C09154=1166.613,121.916,-54.152,-178.809,6.458,148.827
C09155=1166.608,122.166,-54.171,-178.807,6.459,148.826
C09156=1166.603,122.415,-54.191,-178.804,6.460,148.826
C09157=1166.598,122.664,-54.210,-178.801,6.462,148.825
C09158=1166.594,122.914,-54.229,-178.798,6.464,148.825
C09159=1166.589,123.163,-54.249,-178.795,6.466,148.825
C09160=1166.584,123.411,-54.269,-178.793,6.467,148.824
C09161=1166.579,123.661,-54.289,-178.790,6.468,148.824
C09162=1166.575,123.911,-54.308,-178.787,6.470,148.823
C09163=1166.569,124.159,-54.328,-178.785,6.471,148.823
C09164=1166.565,124.409,-54.347,-178.782,6.473,148.822
C09165=1166.561,124.658,-54.367,-178.779,6.475,148.822
C09166=1166.556,124.906,-54.386,-178.777,6.477,148.822
C09167=1166.551,125.156,-54.406,-178.773,6.478,148.821
C09168=1166.546,125.406,-54.426,-178.771,6.479,148.821
C09169=1166.541,125.654,-54.445,-178.769,6.481,148.820
C09170=1166.536,125.903,-54.465,-178.766,6.482,148.820
C09171=1166.532,126.153,-54.485,-178.763,6.484,148.819
C09172=1166.527,126.403,-54.505,-178.760,6.486,148.819
C09173=1166.522,126.651,-54.525,-178.757,6.487,148.818
C09174=1166.517,126.900,-54.544,-178.755,6.488,148.818
C09175=1166.512,127.150,-54.564,-178.752,6.490,148.817
C09176=1166.507,127.399,-54.583,-178.750,6.491,148.817
C09177=1166.502,127.648,-54.604,-178.747,6.493,148.817
C09178=1166.498,127.897,-54.623,-178.744,6.495,148.816
C09179=1166.493,128.147,-54.643,-178.741,6.496,148.816
C09180=1166.488,128.395,-54.663,-178.738,6.498,148.815
C09181=1166.483,128.645,-54.683,-178.736,6.500,148.815
C09182=1166.479,128.894,-54.703,-178.733,6.501,148.814
C09183=1166.474,129.143,-54.723,-178.731,6.502,148.814
C09184=1166.469,129.392,-54.742,-178.728,6.504,148.814
C09185=1166.464,129.641,-54.762,-178.725,6.506,148.813
C09186=1166.460,129.891,-54.782,-178.722,6.507,148.813
C09187=1166.455,130.140,-54.802,-178.719,6.509,148.812
C09188=1166.450,130.389,-54.822,-178.717,6.511,148.812
C09189=1166.445,130.637,-54.842,-178.714,6.512,148.812
C09190=1166.441,130.887,-54.862,-178.712,6.513,148.811
C09191=1166.436,131.136,-54.882,-178.709,6.515,148.811
C09192=1166.431,131.385,-54.902,-178.707,6.517,148.810
C09193=1166.427,131.634,-54.922,-178.704,6.519,148.810
C09194=1166.421,131.903,-54.943,-178.701,6.520,148.809
C09195=1166.416,132.171,-54.965,-178.698,6.522,148.809
C09196=1166.410,132.440,-54.987,-178.695,6.524,148.809
C09197=1166.406,132.708,-55.008,-178.691,6.526,148.808
C09198=1166.401,132.958,-55.028,-178.689,6.527,148.808
C09199=1166.396,133.207,-55.048,-178.687,6.528,148.807
C09200=1166.391,133.456,-55.069,-178.684,6.530,148.807
C09201=1166.386,133.706,-55.089,-178.681,6.532,148.806
C09202=1166.382,133.955,-55.109,-178.679,6.533,148.806
C09203=1166.377,134.204,-55.129,-178.676,6.535,148.806
C09204=1166.372,134.452,-55.149,-178.673,6.537,148.805
C09205=1166.368,134.701,-55.169,-178.670,6.538,148.805
C09206=1166.362,134.951,-55.189,-178.667,6.540,148.804
C09207=1166.358,135.200,-55.210,-178.665,6.542,148.804
C09208=1166.353,135.449,-55.230,-178.662,6.543,148.803
C09209=1166.349,135.699,-55.250,-178.659,6.545,148.803
C09210=1166.344,135.948,-55.270,-178.656,6.547,148.803
C09211=1166.339,136.197,-55.291,-178.654,6.548,148.802
C09212=1166.334,136.446,-55.310,-178.652,6.550,148.802
C09213=1166.329,136.695,-55.331,-178.649,6.551,148.801
C09214=1166.325,136.944,-55.351,-178.646,6.553,148.801
C09215=1166.320,137.193,-55.372,-178.643,6.554,148.800
C09216=1166.315,137.442,-55.392,-178.640,6.556,148.800
C09217=1166.310,137.691,-55.412,-178.638,6.558,148.800
C09218=1166.305,137.941,-55.433,-178.635,6.560,148.799
C09219=1166.301,138.190,-55.453,-178.632,6.561,148.799
C09220=1166.296,138.439,-55.473,-178.629,6.563,148.798
C09221=1166.292,138.688,-55.493,-178.627,6.565,148.798
C09222=1166.287,138.937,-55.514,-178.624,6.567,148.798
C09223=1166.282,139.186,-55.535,-178.621,6.568,148.797
C09224=1166.278,139.435,-55.555,-178.619,6.570,148.797
C09225=1166.272,139.685,-55.576,-178.616,6.572,148.797
C09226=1166.268,139.934,-55.597,-178.613,6.573,148.796
C09227=1166.263,140.183,-55.616,-178.611,6.574,148.796
C09228=1166.258,140.432,-55.637,-178.608,6.576,148.795
C09229=1166.254,140.681,-55.658,-178.605,6.578,148.795
C09230=1166.249,140.930,-55.678,-178.603,6.579,148.794
C09231=1166.244,141.180,-55.699,-178.600,6.581,148.794
C09232=1166.240,141.428,-55.719,-178.597,6.583,148.794
C09233=1166.234,141.678,-55.740,-178.594,6.584,148.793
C09234=1166.230,141.927,-55.761,-178.592,6.586,148.793
C09235=1166.226,142.176,-55.781,-178.589,6.588,148.792
C09236=1166.220,142.425,-55.802,-178.586,6.590,148.792
C09237=1166.216,142.674,-55.822,-178.584,6.591,148.792
C09238=1166.211,142.923,-55.843,-178.581,6.593,148.791
C09239=1166.206,143.172,-55.864,-178.578,6.595,148.791
C09240=1166.202,143.421,-55.884,-178.576,6.597,148.791
C09241=1166.197,143.670,-55.905,-178.573,6.598,148.790
C09242=1166.192,143.919,-55.925,-178.570,6.600,148.790
C09243=1166.187,144.168,-55.946,-178.567,6.601,148.789
C09244=1166.183,144.417,-55.967,-178.564,6.603,148.789
C09245=1166.178,144.667,-55.988,-178.562,6.605,148.788
C09246=1166.173,144.916,-56.008,-178.559,6.607,148.788
C09247=1166.168,145.165,-56.029,-178.556,6.608,148.788
C09248=1166.163,145.414,-56.049,-178.553,6.610,148.787
C09249=1166.158,145.663,-56.070,-178.551,6.612,148.787
C09250=1166.154,145.911,-56.091,-178.548,6.614,148.786
C09251=1166.149,146.161,-56.112,-178.545,6.615,148.786
C09252=1166.145,146.410,-56.133,-178.543,6.617,148.786
C09253=1166.140,146.660,-56.154,-178.540,6.619,148.785
C09254=1166.136,146.909,-56.174,-178.537,6.621,148.785
C09255=1166.130,147.158,-56.195,-178.535,6.622,148.785
C09256=1166.125,147.406,-56.217,-178.532,6.624,148.784
C09257=1166.121,147.655,-56.237,-178.529,6.626,148.784
C09258=1166.116,147.905,-56.258,-178.526,6.628,148.783
C09259=1166.111,148.154,-56.279,-178.524,6.629,148.783
C09260=1166.106,148.403,-56.300,-178.521,6.631,148.783
C09261=1166.102,148.652,-56.322,-178.518,6.633,148.782
C09262=1166.098,148.901,-56.342,-178.516,6.635,148.782
C09263=1166.092,149.150,-56.363,-178.513,6.636,148.781
C09264=1166.088,149.399,-56.384,-178.510,6.638,148.781
C09265=1166.083,149.648,-56.405,-178.508,6.640,148.781
C09266=1166.078,149.897,-56.426,-178.505,6.642,148.780
C09267=1166.073,150.146,-56.447,-178.502,6.643,148.780
C09268=1166.069,150.396,-56.469,-178.499,6.645,148.780
C09269=1166.064,150.645,-56.490,-178.497,6.647,148.779
C09270=1166.060,150.894,-56.510,-178.494,6.648,148.779
C09271=1166.055,151.142,-56.532,-178.491,6.650,148.778
C09272=1166.050,151.392,-56.553,-178.489,6.652,148.778
C09273=1166.045,151.640,-56.574,-178.486,6.654,148.778
C09274=1166.041,151.890,-56.595,-178.483,6.655,148.777
C09275=1166.036,152.139,-56.616,-178.481,6.657,148.777
C09276=1166.031,152.388,-56.638,-178.478,6.659,148.777
C09277=1166.026,152.637,-56.658,-178.475,6.661,148.776
C09278=1166.021,152.885,-56.680,-178.473,6.662,148.776
C09279=1166.017,153.135,-56.701,-178.469,6.665,148.775
C09280=1166.013,153.384,-56.722,-178.467,6.667,148.775
C09281=1166.008,153.633,-56.743,-178.464,6.668,148.775
C09282=1166.002,153.882,-56.764,-178.461,6.670,148.774
C09283=1165.998,154.132,-56.786,-178.458,6.672,148.774
C09284=1165.993,154.381,-56.807,-178.456,6.674,148.774
C09285=1165.989,154.629,-56.828,-178.453,6.675,148.773
C09286=1165.984,154.878,-56.849,-178.450,6.677,148.773
C09287=1165.979,155.128,-56.871,-178.448,6.679,148.772
C09288=1165.975,155.376,-56.893,-178.445,6.681,148.772
C09289=1165.969,155.626,-56.914,-178.442,6.682,148.772
C09290=1165.965,155.874,-56.935,-178.440,6.684,148.771
C09291=1165.961,156.124,-56.956,-178.437,6.686,148.771
C09292=1165.956,156.373,-56.978,-178.434,6.688,148.771
C09293=1165.951,156.622,-56.999,-178.431,6.689,148.770
C09294=1165.946,156.871,-57.021,-178.429,6.691,148.770
C09295=1165.941,157.120,-57.043,-178.426,6.694,148.769
C09296=1165.937,157.369,-57.063,-178.423,6.695,148.769
C09297=1165.932,157.617,-57.085,-178.420,6.697,148.769
C09298=1165.927,157.887,-57.108,-178.417,6.699,148.768
C09299=1165.922,158.155,-57.132,-178.415,6.701,148.768
C09300=1165.917,158.425,-57.155,-178.411,6.703,148.768
C09301=1165.912,158.694,-57.178,-178.409,6.705,148.767
C09302=1165.907,158.942,-57.199,-178.406,6.707,148.767
C09303=1165.903,159.192,-57.221,-178.403,6.709,148.766
C09304=1165.898,159.441,-57.242,-178.401,6.710,148.766
C09305=1165.893,159.690,-57.264,-178.398,6.712,148.766
C09306=1165.889,159.939,-57.286,-178.395,6.714,148.765
C09307=1165.884,160.187,-57.308,-178.392,6.716,148.765
C09308=1165.879,160.437,-57.329,-178.389,6.718,148.765
C09309=1165.874,160.686,-57.351,-178.387,6.720,148.764
C09310=1165.869,160.935,-57.372,-178.384,6.722,148.764
C09311=1165.865,161.184,-57.394,-178.382,6.724,148.764
C09312=1165.860,161.433,-57.416,-178.379,6.725,148.763
C09313=1165.855,161.682,-57.437,-178.376,6.727,148.763
C09314=1165.851,161.931,-57.459,-178.374,6.729,148.763
C09315=1165.846,162.180,-57.481,-178.371,6.731,148.762
C09316=1165.842,162.429,-57.503,-178.368,6.733,148.762
C09317=1165.837,162.678,-57.525,-178.365,6.735,148.761
C09318=1165.833,162.927,-57.547,-178.362,6.737,148.761
C09319=1165.828,163.176,-57.568,-178.360,6.738,148.761
C09320=1165.823,163.425,-57.590,-178.357,6.740,148.760
C09321=1165.819,163.674,-57.612,-178.354,6.742,148.760
C09322=1165.814,163.923,-57.634,-178.352,6.744,148.760
C09323=1165.809,164.172,-57.655,-178.349,6.746,148.759
C09324=1165.804,164.421,-57.677,-178.347,6.748,148.759
C09325=1165.800,164.670,-57.699,-178.343,6.750,148.759
C09326=1165.795,164.919,-57.720,-178.341,6.752,148.758
C09327=1165.790,165.168,-57.742,-178.338,6.754,148.758
C09328=1165.785,165.417,-57.765,-178.335,6.755,148.758
C09329=1165.780,165.666,-57.786,-178.333,6.757,148.757
C09330=1165.776,165.915,-57.809,-178.330,6.759,148.757
C09331=1165.771,166.164,-57.830,-178.327,6.761,148.756
C09332=1165.767,166.413,-57.853,-178.324,6.763,148.756
C09333=1165.762,166.661,-57.875,-178.322,6.765,148.756
C09334=1165.758,166.911,-57.897,-178.319,6.767,148.756
C09335=1165.752,167.160,-57.919,-178.316,6.769,148.755
C09336=1165.748,167.409,-57.941,-178.314,6.771,148.755
C09337=1165.743,167.658,-57.963,-178.311,6.772,148.754
C09338=1165.739,167.907,-57.985,-178.308,6.774,148.754
C09339=1165.734,168.156,-58.006,-178.305,6.777,148.754
C09340=1165.729,168.405,-58.029,-178.302,6.778,148.753
C09341=1165.725,168.653,-58.051,-178.300,6.781,148.753
C09342=1165.720,168.903,-58.074,-178.297,6.782,148.753
C09343=1165.716,169.151,-58.095,-178.295,6.784,148.753
C09344=1165.711,169.401,-58.118,-178.292,6.786,148.752
C09345=1165.706,169.650,-58.140,-178.289,6.788,148.752
C09346=1165.701,169.899,-58.162,-178.286,6.790,148.751
C09347=1165.697,170.148,-58.184,-178.283,6.792,148.751
C09348=1165.692,170.397,-58.207,-178.281,6.794,148.751
C09349=1165.688,170.646,-58.229,-178.279,6.796,148.751
C09350=1165.683,170.895,-58.250,-178.276,6.797,148.750
C09351=1165.679,171.143,-58.273,-178.273,6.800,148.750
C09352=1165.673,171.392,-58.295,-178.270,6.802,148.749
C09353=1165.669,171.642,-58.317,-178.267,6.804,148.749
C09354=1165.665,171.890,-58.340,-178.265,6.805,148.749
C09355=1165.659,172.139,-58.363,-178.262,6.807,148.748
C09356=1165.655,172.389,-58.385,-178.259,6.810,148.748
C09357=1165.650,172.637,-58.407,-178.256,6.812,148.748
C09358=1165.645,172.886,-58.430,-178.254,6.814,148.748
C09359=1165.641,173.136,-58.452,-178.251,6.815,148.747
C09360=1165.637,173.384,-58.474,-178.248,6.817,148.747
C09361=1165.632,173.633,-58.497,-178.245,6.820,148.746
C09362=1165.627,173.882,-58.518,-178.243,6.822,148.746
C09363=1165.622,174.131,-58.542,-178.240,6.823,148.746
C09364=1165.618,174.380,-58.564,-178.237,6.825,148.746
C09365=1165.613,174.628,-58.586,-178.235,6.827,148.745
C09366=1165.608,174.878,-58.609,-178.231,6.830,148.745
C09367=1165.604,175.127,-58.632,-178.229,6.831,148.744
C09368=1165.599,175.376,-58.654,-178.227,6.833,148.744
C09369=1165.595,175.624,-58.677,-178.224,6.835,148.744
C09370=1165.590,175.874,-58.699,-178.221,6.837,148.744
C09371=1165.585,176.123,-58.721,-178.218,6.840,148.743
C09372=1165.581,176.371,-58.744,-178.215,6.841,148.743
C09373=1165.576,176.620,-58.767,-178.213,6.843,148.743
C09374=1165.571,176.869,-58.789,-178.210,6.845,148.742
C09375=1165.567,177.118,-58.812,-178.208,6.847,148.742
C09376=1165.562,177.367,-58.834,-178.204,6.849,148.742
C09377=1165.557,177.616,-58.857,-178.202,6.851,148.741
C09378=1165.553,177.865,-58.879,-178.200,6.853,148.741
C09379=1165.548,178.114,-58.903,-178.197,6.855,148.741
C09380=1165.544,178.363,-58.925,-178.194,6.858,148.740
C09381=1165.538,178.612,-58.948,-178.191,6.859,148.740
C09382=1165.534,178.861,-58.970,-178.188,6.861,148.740
C09383=1165.529,179.110,-58.993,-178.186,6.863,148.740
C09384=1165.525,179.358,-59.015,-178.183,6.866,148.739
C09385=1165.520,179.607,-59.039,-178.180,6.868,148.739
C09386=1165.516,179.857,-59.061,-178.177,6.869,148.739
C09387=1165.511,180.106,-59.084,-178.175,6.871,148.738
C09388=1165.506,180.354,-59.107,-178.172,6.873,148.738
C09389=1165.502,180.603,-59.130,-178.169,6.876,148.738
C09390=1165.497,180.852,-59.153,-178.167,6.878,148.737
C09391=1165.493,181.101,-59.175,-178.164,6.879,148.737
C09392=1165.488,181.350,-59.199,-178.161,6.881,148.737
C09393=1165.483,181.599,-59.221,-178.158,6.884,148.737
C09394=1165.479,181.848,-59.244,-178.156,6.886,148.736
C09395=1165.474,182.097,-59.267,-178.153,6.888,148.736
C09396=1165.470,182.345,-59.290,-178.150,6.889,148.735
C09397=1165.465,182.595,-59.313,-178.148,6.892,148.735
C09398=1165.460,182.843,-59.335,-178.145,6.894,148.735
C09399=1165.456,183.092,-59.358,-178.142,6.896,148.735
C09400=1165.451,183.341,-59.382,-178.139,6.898,148.734
C09401=1165.446,183.590,-59.405,-178.137,6.900,148.734
C09402=1165.442,183.860,-59.429,-178.134,6.902,148.734
C09403=1165.437,184.129,-59.454,-178.131,6.905,148.733
C09404=1165.431,184.399,-59.479,-178.128,6.907,148.733
C09405=1165.427,184.668,-59.505,-178.125,6.909,148.733
C09406=1165.422,184.918,-59.527,-178.122,6.911,148.732
C09407=1165.417,185.167,-59.551,-178.119,6.914,148.732
C09408=1165.412,185.415,-59.574,-178.117,6.916,148.732
C09409=1165.408,185.664,-59.596,-178.114,6.917,148.732
C09410=1165.403,185.913,-59.620,-178.111,6.919,148.731
C09411=1165.399,186.162,-59.643,-178.109,6.922,148.731
C09412=1165.394,186.411,-59.666,-178.106,6.924,148.731
C09413=1165.390,186.660,-59.689,-178.103,6.926,148.730
C09414=1165.385,186.909,-59.713,-178.100,6.928,148.730
C09415=1165.380,187.158,-59.736,-178.098,6.930,148.730
C09416=1165.376,187.407,-59.759,-178.095,6.932,148.730
C09417=1165.370,187.655,-59.782,-178.092,6.934,148.729
C09418=1165.367,187.904,-59.805,-178.089,6.936,148.729
C09419=1165.362,188.153,-59.828,-178.087,6.938,148.729
C09420=1165.357,188.401,-59.853,-178.084,6.940,148.728
C09421=1165.353,188.650,-59.876,-178.081,6.943,148.728
C09422=1165.348,188.899,-59.899,-178.079,6.945,148.728
C09423=1165.343,189.148,-59.923,-178.076,6.947,148.728
C09424=1165.339,189.397,-59.946,-178.073,6.949,148.727
C09425=1165.335,189.646,-59.969,-178.070,6.951,148.727
C09426=1165.330,189.895,-59.992,-178.068,6.953,148.727
C09427=1165.325,190.144,-60.015,-178.065,6.956,148.726
C09428=1165.321,190.393,-60.039,-178.062,6.958,148.726
C09429=1165.316,190.642,-60.063,-178.060,6.960,148.726
C09430=1165.311,190.891,-60.086,-178.057,6.961,148.726
C09431=1165.306,191.139,-60.109,-178.054,6.964,148.725
C09432=1165.301,191.388,-60.133,-178.052,6.966,148.725
C09433=1165.297,191.636,-60.157,-178.049,6.968,148.725
C09434=1165.292,191.885,-60.180,-178.046,6.970,148.724
C09435=1165.288,192.134,-60.203,-178.043,6.972,148.724
C09436=1165.283,192.383,-60.227,-178.041,6.974,148.724
C09437=1165.279,192.632,-60.251,-178.038,6.977,148.724
C09438=1165.274,192.881,-60.274,-178.035,6.979,148.723
C09439=1165.269,193.130,-60.298,-178.033,6.981,148.723
C09440=1165.265,193.378,-60.322,-178.029,6.983,148.723
C09441=1165.260,193.627,-60.345,-178.027,6.985,148.722
C09442=1165.255,193.876,-60.368,-178.025,6.987,148.722
C09443=1165.251,194.125,-60.392,-178.021,6.990,148.722
C09444=1165.246,194.374,-60.416,-178.019,6.992,148.722
C09445=1165.242,194.624,-60.439,-178.016,6.995,148.721
C09446=1165.238,194.872,-60.464,-178.013,6.996,148.721
C09447=1165.233,195.121,-60.487,-178.010,6.998,148.721
C09448=1165.229,195.369,-60.511,-178.008,7.001,148.721
C09449=1165.224,195.619,-60.534,-178.005,7.003,148.720
C09450=1165.219,195.868,-60.558,-178.002,7.005,148.720
C09451=1165.215,196.116,-60.582,-178.000,7.007,148.720
C09452=1165.210,196.365,-60.605,-177.997,7.009,148.720
C09453=1165.206,196.613,-60.629,-177.994,7.011,148.719
C09454=1165.201,196.862,-60.653,-177.991,7.014,148.719
C09455=1165.197,197.111,-60.677,-177.989,7.016,148.719
C09456=1165.191,197.360,-60.701,-177.987,7.018,148.719
C09457=1165.187,197.609,-60.725,-177.983,7.020,148.718
C09458=1165.182,197.858,-60.748,-177.981,7.022,148.718
C09459=1165.178,198.107,-60.772,-177.978,7.025,148.718
C09460=1165.174,198.356,-60.796,-177.975,7.027,148.717
C09461=1165.169,198.604,-60.820,-177.972,7.029,148.717
C09462=1165.165,198.853,-60.844,-177.970,7.032,148.717
C09463=1165.159,199.102,-60.868,-177.967,7.033,148.717
C09464=1165.155,199.350,-60.892,-177.964,7.035,148.716
C09465=1165.150,199.599,-60.915,-177.962,7.038,148.716
C09466=1165.147,199.849,-60.940,-177.959,7.040,148.716
C09467=1165.142,200.097,-60.964,-177.956,7.043,148.716
C09468=1165.137,200.346,-60.988,-177.953,7.045,148.715
C09469=1165.132,200.595,-61.012,-177.951,7.046,148.715
C09470=1165.128,200.843,-61.036,-177.948,7.049,148.715
C09471=1165.123,201.092,-61.059,-177.945,7.051,148.715
C09472=1165.119,201.342,-61.084,-177.943,7.054,148.715
C09473=1165.114,201.590,-61.108,-177.940,7.056,148.714
C09474=1165.110,201.839,-61.132,-177.937,7.058,148.714
C09475=1165.105,202.087,-61.156,-177.934,7.060,148.714
C09476=1165.100,202.336,-61.181,-177.932,7.062,148.713
C09477=1165.096,202.585,-61.205,-177.928,7.065,148.713
C09478=1165.092,202.834,-61.229,-177.926,7.067,148.713
C09479=1165.087,203.083,-61.252,-177.924,7.069,148.713
C09480=1165.082,203.331,-61.277,-177.921,7.072,148.712
C09481=1165.078,203.580,-61.301,-177.918,7.073,148.712
C09482=1165.074,203.829,-61.326,-177.915,7.076,148.712
C09483=1165.069,204.078,-61.350,-177.913,7.078,148.712
C09484=1165.064,204.327,-61.374,-177.909,7.081,148.711
C09485=1165.060,204.575,-61.398,-177.907,7.083,148.711
C09486=1165.055,204.825,-61.423,-177.905,7.085,148.711
C09487=1165.051,205.073,-61.447,-177.902,7.088,148.711
C09488=1165.046,205.321,-61.471,-177.899,7.089,148.710
C09489=1165.041,205.570,-61.496,-177.896,7.092,148.710
C09490=1165.037,205.819,-61.520,-177.894,7.094,148.710
C09491=1165.032,206.068,-61.545,-177.891,7.096,148.710
C09492=1165.028,206.316,-61.569,-177.888,7.099,148.710
C09493=1165.023,206.565,-61.593,-177.886,7.101,148.709
C09494=1165.019,206.814,-61.618,-177.883,7.103,148.709
C09495=1165.015,207.063,-61.642,-177.880,7.105,148.709
C09496=1165.009,207.311,-61.667,-177.877,7.108,148.708
C09497=1165.006,207.560,-61.691,-177.875,7.110,148.708
C09498=1165.001,207.809,-61.716,-177.871,7.113,148.708
C09499=1164.996,208.058,-61.740,-177.869,7.115,148.708
C09500=1164.991,208.306,-61.764,-177.867,7.116,148.708
C09501=1164.987,208.555,-61.789,-177.864,7.119,148.707
C09502=1164.982,208.804,-61.814,-177.861,7.121,148.707
C09503=1164.978,209.053,-61.838,-177.858,7.124,148.707
C09504=1164.973,209.302,-61.863,-177.856,7.126,148.707
C09505=1164.969,209.550,-61.887,-177.853,7.129,148.707
C09506=1164.964,209.821,-61.913,-177.850,7.131,148.706
C09507=1164.959,210.091,-61.941,-177.847,7.133,148.706
C09508=1164.954,210.362,-61.967,-177.844,7.136,148.706
C09509=1164.949,210.632,-61.994,-177.841,7.139,148.705
C09510=1164.944,210.881,-62.019,-177.838,7.140,148.705
C09511=1164.940,211.130,-62.043,-177.836,7.143,148.705
C09512=1164.935,211.379,-62.068,-177.833,7.145,148.705
C09513=1164.931,211.627,-62.092,-177.830,7.148,148.705
C09514=1164.927,211.876,-62.118,-177.827,7.150,148.704
C09515=1164.922,212.125,-62.143,-177.825,7.153,148.704
C09516=1164.917,212.373,-62.167,-177.822,7.155,148.704
C09517=1164.913,212.623,-62.192,-177.819,7.158,148.704
C09518=1164.909,212.871,-62.216,-177.817,7.159,148.703
C09519=1164.904,213.120,-62.242,-177.814,7.162,148.703
C09520=1164.899,213.369,-62.266,-177.811,7.164,148.703
C09521=1164.894,213.617,-62.290,-177.809,7.166,148.703
C09522=1164.890,213.866,-62.316,-177.806,7.169,148.703
C09523=1164.885,214.115,-62.341,-177.803,7.171,148.702
C09524=1164.881,214.364,-62.365,-177.800,7.174,148.702
C09525=1164.877,214.612,-62.391,-177.798,7.176,148.702
C09526=1164.872,214.861,-62.416,-177.795,7.178,148.702
C09527=1164.868,215.110,-62.440,-177.793,7.180,148.702
C09528=1164.863,215.359,-62.465,-177.789,7.183,148.701
C09529=1164.858,215.607,-62.490,-177.787,7.185,148.701
C09530=1164.853,215.855,-62.515,-177.784,7.188,148.701
C09531=1164.850,216.104,-62.540,-177.782,7.190,148.701
C09532=1164.845,216.353,-62.565,-177.778,7.192,148.700
C09533=1164.840,216.602,-62.590,-177.776,7.194,148.700
C09534=1164.835,216.851,-62.615,-177.773,7.197,148.700
C09535=1164.832,217.099,-62.640,-177.770,7.200,148.700
C09536=1164.827,217.348,-62.665,-177.768,7.202,148.700
C09537=1164.822,217.597,-62.691,-177.765,7.205,148.699
C09538=1164.817,217.845,-62.715,-177.762,7.207,148.699
C09539=1164.814,218.094,-62.740,-177.759,7.209,148.699
C09540=1164.809,218.343,-62.765,-177.757,7.211,148.699
C09541=1164.804,218.591,-62.791,-177.754,7.214,148.699
C09542=1164.800,218.840,-62.817,-177.752,7.216,148.698
C09543=1164.795,219.089,-62.841,-177.748,7.219,148.698
C09544=1164.791,219.338,-62.866,-177.746,7.221,148.698
C09545=1164.786,219.586,-62.891,-177.743,7.224,148.698
C09546=1164.782,219.835,-62.917,-177.741,7.226,148.698
C09547=1164.777,220.083,-62.942,-177.738,7.228,148.697
C09548=1164.773,220.333,-62.967,-177.735,7.230,148.697
C09549=1164.768,220.581,-62.993,-177.732,7.233,148.697
C09550=1164.764,220.829,-63.018,-177.730,7.235,148.697
C09551=1164.760,221.079,-63.043,-177.727,7.238,148.697
C09552=1164.755,221.327,-63.068,-177.724,7.241,148.696
C09553=1164.751,221.575,-63.094,-177.722,7.243,148.696
C09554=1164.746,221.824,-63.119,-177.718,7.245,148.696
C09555=1164.742,222.073,-63.144,-177.716,7.248,148.696
C09556=1164.737,222.322,-63.170,-177.713,7.250,148.696
C09557=1164.732,222.570,-63.195,-177.711,7.252,148.695
C09558=1164.728,222.819,-63.221,-177.708,7.255,148.695
C09559=1164.723,223.067,-63.246,-177.705,7.257,148.695
C09560=1164.719,223.316,-63.272,-177.703,7.260,148.695
C09561=1164.715,223.565,-63.297,-177.699,7.263,148.695
C09562=1164.710,223.814,-63.322,-177.697,7.265,148.695
C09563=1164.705,224.063,-63.348,-177.694,7.267,148.694
C09564=1164.701,224.311,-63.374,-177.692,7.269,148.694
C09565=1164.696,224.560,-63.399,-177.689,7.272,148.694
C09566=1164.692,224.808,-63.425,-177.686,7.274,148.694
C09567=1164.687,225.056,-63.450,-177.684,7.277,148.694
C09568=1164.683,225.305,-63.476,-177.680,7.280,148.693
C09569=1164.678,225.555,-63.501,-177.678,7.282,148.693
C09570=1164.674,225.803,-63.526,-177.675,7.285,148.693
C09571=1164.669,226.052,-63.552,-177.673,7.287,148.693
C09572=1164.665,226.300,-63.578,-177.670,7.290,148.693
C09573=1164.661,226.549,-63.604,-177.667,7.291,148.692
C09574=1164.656,226.797,-63.629,-177.665,7.294,148.692
C09575=1164.652,227.046,-63.655,-177.662,7.297,148.692
C09576=1164.648,227.295,-63.680,-177.659,7.299,148.692
C09577=1164.642,227.543,-63.706,-177.656,7.302,148.692
C09578=1164.638,227.792,-63.732,-177.654,7.304,148.692
C09579=1164.634,228.041,-63.758,-177.651,7.307,148.691
C09580=1164.629,228.290,-63.784,-177.648,7.310,148.691
C09581=1164.625,228.538,-63.809,-177.645,7.311,148.691
C09582=1164.620,228.787,-63.835,-177.643,7.314,148.691
C09583=1164.616,229.035,-63.861,-177.640,7.316,148.691
C09584=1164.611,229.284,-63.886,-177.637,7.319,148.690
C09585=1164.607,229.532,-63.913,-177.634,7.322,148.690
C09586=1164.602,229.781,-63.939,-177.632,7.324,148.690
C09587=1164.598,230.030,-63.964,-177.629,7.327,148.690
C09588=1164.594,230.278,-63.990,-177.626,7.330,148.690
C09589=1164.588,230.527,-64.016,-177.624,7.332,148.690
C09590=1164.584,230.776,-64.042,-177.621,7.334,148.689
C09591=1164.580,231.024,-64.068,-177.619,7.337,148.689
C09592=1164.576,231.273,-64.094,-177.615,7.339,148.689
C09593=1164.571,231.521,-64.120,-177.613,7.342,148.689
C09594=1164.566,231.770,-64.146,-177.610,7.344,148.689
C09595=1164.562,232.019,-64.172,-177.607,7.347,148.689
C09596=1164.558,232.267,-64.197,-177.604,7.350,148.689
C09597=1164.554,232.516,-64.224,-177.602,7.352,148.688
C09598=1164.548,232.764,-64.250,-177.599,7.355,148.688
C09599=1164.544,233.013,-64.276,-177.597,7.357,148.688
C09600=1164.540,233.261,-64.302,-177.594,7.360,148.688
C09601=1164.535,233.510,-64.328,-177.591,7.363,148.688
C09602=1164.531,233.759,-64.354,-177.589,7.364,148.688
C09603=1164.527,234.008,-64.380,-177.586,7.367,148.687
C09604=1164.522,234.256,-64.407,-177.583,7.370,148.687
C09605=1164.517,234.504,-64.432,-177.580,7.372,148.687
C09606=1164.513,234.753,-64.459,-177.578,7.375,148.687
C09607=1164.508,235.002,-64.485,-177.575,7.378,148.687
C09608=1164.504,235.250,-64.511,-177.572,7.380,148.687
C09609=1164.500,235.499,-64.537,-177.570,7.383,148.686
C09610=1164.495,235.771,-64.566,-177.567,7.386,148.686
C09611=1164.490,236.042,-64.595,-177.564,7.388,148.686
C09612=1164.485,236.314,-64.623,-177.561,7.391,148.686
C09613=1164.481,236.586,-64.652,-177.558,7.394,148.686
C09614=1164.476,236.835,-64.679,-177.555,7.397,148.686
C09615=1164.472,237.083,-64.705,-177.553,7.399,148.686
C09616=1164.467,237.331,-64.730,-177.550,7.402,148.685
C09617=1164.462,237.580,-64.757,-177.547,7.404,148.685
C09618=1164.458,237.828,-64.783,-177.544,7.407,148.685
C09619=1164.453,238.077,-64.810,-177.542,7.409,148.685
C09620=1164.449,238.326,-64.836,-177.538,7.412,148.685
C09621=1164.445,238.574,-64.863,-177.536,7.414,148.685
C09622=1164.441,238.822,-64.890,-177.533,7.417,148.685
C09623=1164.436,239.071,-64.916,-177.531,7.420,148.684
C09624=1164.432,239.320,-64.942,-177.528,7.422,148.684
C09625=1164.427,239.569,-64.969,-177.525,7.425,148.684
C09626=1164.423,239.817,-64.995,-177.522,7.428,148.684
C09627=1164.418,240.065,-65.022,-177.520,7.430,148.684
C09628=1164.414,240.314,-65.048,-177.517,7.433,148.684
C09629=1164.409,240.563,-65.075,-177.514,7.435,148.684
C09630=1164.405,240.811,-65.101,-177.512,7.438,148.683
C09631=1164.400,241.060,-65.128,-177.509,7.441,148.683
C09632=1164.396,241.309,-65.155,-177.506,7.443,148.683
C09633=1164.392,241.557,-65.181,-177.503,7.446,148.683
C09634=1164.387,241.806,-65.208,-177.501,7.448,148.683
C09635=1164.383,242.054,-65.234,-177.498,7.451,148.683
C09636=1164.378,242.303,-65.261,-177.496,7.454,148.683
C09637=1164.374,242.551,-65.288,-177.493,7.456,148.682
C09638=1164.370,242.799,-65.315,-177.490,7.459,148.682
C09639=1164.365,243.048,-65.341,-177.487,7.462,148.682
C09640=1164.361,243.297,-65.368,-177.485,7.465,148.682
C09641=1164.356,243.545,-65.395,-177.482,7.467,148.682
C09642=1164.352,243.793,-65.422,-177.479,7.470,148.682
C09643=1164.348,244.042,-65.448,-177.476,7.473,148.682
C09644=1164.343,244.291,-65.474,-177.474,7.475,148.682
C09645=1164.338,244.539,-65.502,-177.472,7.478,148.682
C09646=1164.334,244.787,-65.528,-177.468,7.480,148.681
C09647=1164.329,245.036,-65.555,-177.466,7.483,148.681
C09648=1164.325,245.284,-65.582,-177.463,7.485,148.681
C09649=1164.321,245.533,-65.609,-177.461,7.488,148.681
C09650=1164.317,245.782,-65.636,-177.458,7.491,148.681
C09651=1164.312,246.030,-65.663,-177.455,7.494,148.681
C09652=1164.307,246.279,-65.690,-177.452,7.496,148.681
C09653=1164.304,246.527,-65.717,-177.450,7.499,148.681
C09654=1164.299,246.776,-65.744,-177.447,7.502,148.680
C09655=1164.294,247.024,-65.771,-177.445,7.504,148.680
C09656=1164.290,247.273,-65.798,-177.442,7.507,148.680
C09657=1164.286,247.521,-65.824,-177.439,7.510,148.680
C09658=1164.281,247.769,-65.851,-177.436,7.512,148.680
C09659=1164.277,248.018,-65.879,-177.434,7.515,148.680
C09660=1164.272,248.267,-65.906,-177.431,7.518,148.680
C09661=1164.268,248.515,-65.933,-177.428,7.521,148.680
C09662=1164.264,248.764,-65.959,-177.425,7.523,148.680
C09663=1164.259,249.012,-65.986,-177.423,7.525,148.679
C09664=1164.254,249.261,-66.013,-177.420,7.528,148.679
C09665=1164.250,249.509,-66.041,-177.417,7.531,148.679
C09666=1164.246,249.758,-66.069,-177.415,7.534,148.679
C09667=1164.241,250.006,-66.096,-177.412,7.536,148.679
C09668=1164.237,250.255,-66.123,-177.410,7.539,148.679
C09669=1164.233,250.503,-66.149,-177.407,7.542,148.679
C09670=1164.228,250.751,-66.176,-177.404,7.545,148.679
C09671=1164.224,251.000,-66.204,-177.401,7.548,148.679
C09672=1164.220,251.248,-66.232,-177.399,7.550,148.678
C09673=1164.215,251.497,-66.259,-177.396,7.553,148.678
C09674=1164.210,251.745,-66.286,-177.393,7.556,148.678
C09675=1164.206,251.994,-66.313,-177.390,7.559,148.678
C09676=1164.202,252.242,-66.341,-177.388,7.561,148.678
C09677=1164.197,252.491,-66.368,-177.385,7.564,148.678
C09678=1164.193,252.739,-66.395,-177.382,7.566,148.678
C09679=1164.188,252.988,-66.422,-177.379,7.569,148.678
C09680=1164.184,253.236,-66.450,-177.377,7.571,148.678
C09681=1164.180,253.485,-66.477,-177.374,7.574,148.678
C09682=1164.175,253.733,-66.504,-177.372,7.577,148.678
C09683=1164.171,253.981,-66.532,-177.369,7.580,148.677
C09684=1164.167,254.231,-66.560,-177.366,7.583,148.677
C09685=1164.162,254.478,-66.587,-177.364,7.585,148.677
C09686=1164.158,254.727,-66.614,-177.361,7.588,148.677
C09687=1164.153,254.975,-66.641,-177.358,7.591,148.677
C09688=1164.149,255.224,-66.670,-177.355,7.594,148.677
C09689=1164.144,255.472,-66.697,-177.352,7.597,148.677
C09690=1164.140,255.720,-66.724,-177.350,7.599,148.677
C09691=1164.136,255.970,-66.752,-177.348,7.602,148.677
C09692=1164.132,256.217,-66.780,-177.345,7.605,148.677
C09693=1164.127,256.466,-66.807,-177.342,7.608,148.677
C09694=1164.123,256.715,-66.835,-177.339,7.611,148.677
C09695=1164.119,256.963,-66.862,-177.337,7.613,148.676
C09696=1164.114,257.211,-66.890,-177.334,7.616,148.676
C09697=1164.109,257.460,-66.918,-177.332,7.619,148.676
C09698=1164.105,257.708,-66.945,-177.329,7.622,148.676
C09699=1164.100,257.957,-66.973,-177.326,7.625,148.676
C09700=1164.097,258.205,-67.001,-177.324,7.627,148.676
C09701=1164.092,258.453,-67.028,-177.321,7.630,148.676
C09702=1164.088,258.702,-67.055,-177.318,7.633,148.676
C09703=1164.084,258.950,-67.084,-177.316,7.636,148.676
C09704=1164.079,259.199,-67.111,-177.312,7.638,148.676
C09705=1164.074,259.447,-67.139,-177.310,7.641,148.676
C09706=1164.070,259.696,-67.167,-177.307,7.644,148.675
C09707=1164.066,259.944,-67.194,-177.305,7.646,148.675
C09708=1164.062,260.193,-67.222,-177.302,7.649,148.675
C09709=1164.057,260.441,-67.251,-177.299,7.652,148.675
C09710=1164.052,260.689,-67.278,-177.296,7.655,148.675
C09711=1164.049,260.938,-67.306,-177.294,7.657,148.675
C09712=1164.044,261.186,-67.334,-177.291,7.660,148.675
C09713=1164.040,261.435,-67.363,-177.289,7.663,148.675
C09714=1164.034,261.707,-67.393,-177.286,7.666,148.675
C09715=1164.030,261.981,-67.423,-177.283,7.670,148.675
C09716=1164.025,262.254,-67.454,-177.280,7.673,148.675
C09717=1164.020,262.527,-67.485,-177.277,7.676,148.675
C09718=1164.016,262.775,-67.513,-177.274,7.679,148.675
C09719=1164.012,263.024,-67.541,-177.272,7.682,148.675
C09720=1164.007,263.272,-67.569,-177.269,7.685,148.675
C09721=1164.003,263.521,-67.597,-177.267,7.687,148.675
C09722=1163.999,263.769,-67.624,-177.264,7.690,148.675
C09723=1163.994,264.018,-67.653,-177.261,7.693,148.674
C09724=1163.990,264.266,-67.681,-177.258,7.696,148.674
C09725=1163.986,264.515,-67.710,-177.256,7.699,148.674
C09726=1163.981,264.763,-67.737,-177.253,7.702,148.674
C09727=1163.977,265.011,-67.766,-177.250,7.705,148.674
C09728=1163.972,265.259,-67.794,-177.248,7.707,148.674
C09729=1163.969,265.508,-67.822,-177.245,7.710,148.674
C09730=1163.964,265.756,-67.850,-177.242,7.713,148.674
C09731=1163.960,266.005,-67.879,-177.240,7.716,148.674
C09732=1163.955,266.252,-67.906,-177.237,7.719,148.674
C09733=1163.951,266.501,-67.935,-177.234,7.722,148.674
C09734=1163.947,266.749,-67.963,-177.231,7.725,148.674
C09735=1163.942,266.998,-67.992,-177.229,7.727,148.674
C09736=1163.938,267.246,-68.019,-177.226,7.730,148.674
C09737=1163.933,267.495,-68.048,-177.224,7.733,148.674
C09738=1163.929,267.743,-68.076,-177.221,7.736,148.674
C09739=1163.924,267.992,-68.105,-177.218,7.739,148.674
C09740=1163.920,268.240,-68.132,-177.215,7.742,148.674
C09741=1163.916,268.488,-68.161,-177.213,7.745,148.674
C09742=1163.912,268.737,-68.189,-177.210,7.748,148.674
C09743=1163.907,268.985,-68.218,-177.208,7.750,148.674
C09744=1163.903,269.233,-68.246,-177.205,7.753,148.673
C09745=1163.898,269.481,-68.275,-177.203,7.756,148.673
C09746=1163.894,269.730,-68.303,-177.200,7.759,148.673
C09747=1163.889,269.978,-68.331,-177.197,7.762,148.673
C09748=1163.886,270.226,-68.360,-177.194,7.765,148.673
C09749=1163.881,270.475,-68.389,-177.192,7.768,148.673
C09750=1163.877,270.723,-68.417,-177.189,7.771,148.673
C09751=1163.873,270.972,-68.445,-177.186,7.774,148.673
C09752=1163.868,271.220,-68.475,-177.184,7.776,148.673
C09753=1163.864,271.468,-68.503,-177.182,7.779,148.673
C09754=1163.860,271.717,-68.531,-177.179,7.782,148.673
C09755=1163.855,271.965,-68.559,-177.176,7.785,148.673
C09756=1163.851,272.213,-68.589,-177.173,7.788,148.673
C09757=1163.847,272.462,-68.617,-177.171,7.791,148.673
C09758=1163.842,272.710,-68.645,-177.168,7.794,148.673
C09759=1163.838,272.958,-68.675,-177.165,7.797,148.673
C09760=1163.834,273.207,-68.703,-177.162,7.800,148.673
C09761=1163.830,273.454,-68.732,-177.160,7.803,148.673
C09762=1163.825,273.703,-68.761,-177.158,7.805,148.673
C09763=1163.821,273.952,-68.789,-177.155,7.808,148.673
C09764=1163.817,274.199,-68.818,-177.152,7.811,148.673
C09765=1163.812,274.448,-68.847,-177.150,7.814,148.673
C09766=1163.808,274.696,-68.876,-177.147,7.817,148.673
C09767=1163.803,274.944,-68.904,-177.144,7.820,148.673
C09768=1163.799,275.192,-68.933,-177.141,7.823,148.673
C09769=1163.795,275.441,-68.962,-177.139,7.826,148.673
C09770=1163.791,275.690,-68.991,-177.136,7.829,148.673
C09771=1163.786,275.937,-69.019,-177.133,7.832,148.673
C09772=1163.782,276.186,-69.049,-177.131,7.835,148.673
C09773=1163.778,276.435,-69.077,-177.128,7.838,148.673
C09774=1163.773,276.683,-69.107,-177.126,7.840,148.673
C09775=1163.769,276.931,-69.135,-177.123,7.843,148.673
C09776=1163.765,277.179,-69.164,-177.120,7.846,148.672
C09777=1163.761,277.427,-69.194,-177.118,7.849,148.673
C09778=1163.756,277.676,-69.222,-177.115,7.852,148.673
C09779=1163.751,277.924,-69.251,-177.112,7.855,148.673
C09780=1163.748,278.172,-69.280,-177.110,7.858,148.672
C09781=1163.744,278.421,-69.309,-177.107,7.861,148.672
C09782=1163.739,278.669,-69.338,-177.105,7.865,148.673
C09783=1163.735,278.917,-69.368,-177.102,7.867,148.673
C09784=1163.730,279.165,-69.396,-177.099,7.870,148.673
C09785=1163.726,279.414,-69.426,-177.096,7.873,148.672
C09786=1163.722,279.662,-69.455,-177.094,7.876,148.672
C09787=1163.718,279.910,-69.483,-177.091,7.879,148.672
C09788=1163.714,280.159,-69.513,-177.089,7.883,148.673
C09789=1163.709,280.406,-69.542,-177.086,7.885,148.672
C09790=1163.705,280.654,-69.571,-177.084,7.888,148.672
C09791=1163.700,280.903,-69.600,-177.081,7.891,148.672
C09792=1163.696,281.152,-69.630,-177.078,7.894,148.672
C09793=1163.692,281.400,-69.659,-177.076,7.897,148.673
C09794=1163.688,281.648,-69.688,-177.073,7.900,148.672
C09795=1163.683,281.896,-69.718,-177.070,7.903,148.672
C09796=1163.679,282.144,-69.747,-177.068,7.906,148.672
C09797=1163.674,282.393,-69.776,-177.065,7.909,148.672
C09798=1163.670,282.641,-69.805,-177.063,7.912,148.673
C09799=1163.666,282.889,-69.835,-177.060,7.915,148.672
C09800=1163.662,283.138,-69.864,-177.057,7.918,148.672
C09801=1163.658,283.386,-69.894,-177.054,7.921,148.672
C09802=1163.653,283.634,-69.923,-177.052,7.924,148.673
C09803=1163.649,283.882,-69.952,-177.049,7.927,148.673
C09804=1163.644,284.130,-69.982,-177.046,7.930,148.672
C09805=1163.640,284.378,-70.011,-177.044,7.933,148.672
C09806=1163.636,284.627,-70.040,-177.041,7.936,148.673
C09807=1163.632,284.875,-70.070,-177.039,7.939,148.673
C09808=1163.628,285.123,-70.099,-177.036,7.942,148.673
C09809=1163.624,285.371,-70.129,-177.033,7.945,148.673
C09810=1163.619,285.620,-70.158,-177.031,7.949,148.673
C09811=1163.615,285.868,-70.188,-177.028,7.952,148.673
C09812=1163.610,286.116,-70.217,-177.025,7.955,148.673
C09813=1163.605,286.364,-70.247,-177.023,7.957,148.673
C09814=1163.601,286.612,-70.276,-177.020,7.961,148.673
C09815=1163.597,286.861,-70.306,-177.018,7.964,148.673
C09816=1163.593,287.109,-70.335,-177.015,7.967,148.673
C09817=1163.589,287.357,-70.365,-177.012,7.970,148.673
C09818=1163.584,287.632,-70.398,-177.010,7.973,148.673
C09819=1163.579,287.907,-70.431,-177.007,7.976,148.673
C09820=1163.575,288.182,-70.464,-177.004,7.980,148.673
C09821=1163.570,288.457,-70.497,-177.001,7.983,148.673
C09822=1163.566,288.705,-70.527,-176.999,7.986,148.673
C09823=1163.562,288.953,-70.556,-176.996,7.989,148.673
C09824=1163.557,289.202,-70.586,-176.993,7.992,148.673
C09825=1163.553,289.450,-70.616,-176.990,7.995,148.673
C09826=1163.549,289.698,-70.646,-176.988,7.998,148.673
C09827=1163.544,289.946,-70.675,-176.985,8.001,148.673
C09828=1163.540,290.194,-70.705,-176.983,8.004,148.673
C09829=1163.536,290.442,-70.735,-176.980,8.007,148.673
C09830=1163.531,290.691,-70.765,-176.978,8.010,148.673
C09831=1163.527,290.939,-70.794,-176.975,8.013,148.673
C09832=1163.523,291.186,-70.825,-176.972,8.017,148.673
C09833=1163.518,291.435,-70.855,-176.970,8.020,148.673
C09834=1163.514,291.683,-70.884,-176.967,8.022,148.673
C09835=1163.510,291.931,-70.914,-176.965,8.026,148.673
C09836=1163.506,292.180,-70.945,-176.962,8.029,148.673
C09837=1163.502,292.428,-70.975,-176.959,8.032,148.673
C09838=1163.498,292.676,-71.004,-176.957,8.035,148.673
C09839=1163.493,292.925,-71.034,-176.954,8.038,148.673
C09840=1163.489,293.172,-71.064,-176.951,8.041,148.673
C09841=1163.485,293.421,-71.094,-176.949,8.044,148.674
C09842=1163.480,293.669,-71.125,-176.946,8.047,148.673
C09843=1163.476,293.917,-71.154,-176.944,8.050,148.673
C09844=1163.472,294.165,-71.184,-176.941,8.053,148.674
C09845=1163.467,294.413,-71.214,-176.938,8.057,148.674
C09846=1163.464,294.661,-71.245,-176.935,8.060,148.674
C09847=1163.460,294.910,-71.274,-176.933,8.063,148.674
C09848=1163.455,295.158,-71.305,-176.930,8.066,148.674
C09849=1163.451,295.405,-71.335,-176.927,8.069,148.674
C09850=1163.447,295.654,-71.365,-176.925,8.073,148.674
C09851=1163.443,295.902,-71.395,-176.922,8.076,148.674
C09852=1163.438,296.150,-71.426,-176.920,8.079,148.674
C09853=1163.434,296.399,-71.456,-176.917,8.082,148.674
C09854=1163.430,296.646,-71.487,-176.915,8.085,148.674
C09855=1163.426,296.895,-71.516,-176.912,8.088,148.674
C09856=1163.422,297.142,-71.546,-176.910,8.091,148.674
C09857=1163.417,297.390,-71.577,-176.907,8.094,148.674
C09858=1163.412,297.639,-71.607,-176.904,8.097,148.674
C09859=1163.409,297.887,-71.638,-176.902,8.100,148.674
C09860=1163.404,298.135,-71.669,-176.899,8.104,148.674
C09861=1163.401,298.383,-71.699,-176.897,8.107,148.674
C09862=1163.396,298.631,-71.729,-176.894,8.110,148.674
C09863=1163.392,298.879,-71.759,-176.892,8.113,148.675
C09864=1163.388,299.128,-71.790,-176.889,8.116,148.675
C09865=1163.384,299.375,-71.820,-176.887,8.119,148.675
C09866=1163.379,299.624,-71.850,-176.884,8.122,148.675
C09867=1163.375,299.872,-71.880,-176.881,8.125,148.675
C09868=1163.370,300.120,-71.911,-176.879,8.128,148.675
C09869=1163.366,300.368,-71.942,-176.875,8.132,148.675
C09870=1163.363,300.616,-71.972,-176.873,8.135,148.675
C09871=1163.358,300.864,-72.003,-176.870,8.138,148.675
C09872=1163.353,301.112,-72.033,-176.868,8.142,148.675
C09873=1163.350,301.361,-72.064,-176.865,8.145,148.675
C09874=1163.345,301.609,-72.095,-176.863,8.148,148.675
C09875=1163.341,301.856,-72.125,-176.860,8.151,148.675
C09876=1163.337,302.104,-72.156,-176.858,8.154,148.675
C09877=1163.333,302.353,-72.187,-176.855,8.157,148.675
C09878=1163.328,302.601,-72.217,-176.853,8.160,148.675
C09879=1163.324,302.849,-72.248,-176.850,8.163,148.676
C09880=1163.320,303.097,-72.279,-176.847,8.166,148.676
C09881=1163.316,303.345,-72.309,-176.845,8.170,148.676
C09882=1163.312,303.593,-72.340,-176.842,8.173,148.676
C09883=1163.307,303.841,-72.370,-176.840,8.176,148.676
C09884=1163.303,304.089,-72.402,-176.837,8.180,148.676
C09885=1163.298,304.337,-72.432,-176.834,8.183,148.676
C09886=1163.295,304.585,-72.462,-176.832,8.186,148.676
C09887=1163.291,304.834,-72.494,-176.829,8.189,148.676
C09888=1163.286,305.082,-72.524,-176.827,8.192,148.676
C09889=1163.282,305.329,-72.556,-176.824,8.195,148.676
C09890=1163.278,305.577,-72.586,-176.822,8.198,148.676
C09891=1163.274,305.825,-72.617,-176.819,8.201,148.676
C09892=1163.269,306.073,-72.648,-176.817,8.205,148.677
C09893=1163.265,306.322,-72.679,-176.814,8.208,148.677
C09894=1163.260,306.570,-72.710,-176.812,8.211,148.677
C09895=1163.256,306.819,-72.741,-176.808,8.215,148.677
C09896=1163.253,307.066,-72.772,-176.806,8.218,148.677
C09897=1163.248,307.314,-72.803,-176.803,8.221,148.677
C09898=1163.244,307.562,-72.834,-176.801,8.224,148.677
C09899=1163.240,307.810,-72.864,-176.798,8.227,148.677
C09900=1163.235,308.058,-72.896,-176.796,8.231,148.677
C09901=1163.231,308.306,-72.927,-176.793,8.233,148.677
C09902=1163.227,308.554,-72.958,-176.791,8.237,148.677
C09903=1163.223,308.802,-72.990,-176.788,8.240,148.677
C09904=1163.219,309.050,-73.020,-176.786,8.243,148.678
C09905=1163.215,309.298,-73.051,-176.782,8.247,148.678
C09906=1163.211,309.546,-73.082,-176.780,8.250,148.678
C09907=1163.206,309.794,-73.113,-176.777,8.253,148.678
C09908=1163.202,310.042,-73.144,-176.775,8.256,148.678
C09909=1163.198,310.290,-73.176,-176.773,8.260,148.678
C09910=1163.194,310.538,-73.207,-176.770,8.263,148.678
C09911=1163.189,310.786,-73.238,-176.768,8.266,148.678
C09912=1163.186,311.034,-73.270,-176.765,8.269,148.678
C09913=1163.181,311.282,-73.300,-176.763,8.272,148.679
C09914=1163.177,311.530,-73.332,-176.759,8.276,148.679
C09915=1163.173,311.778,-73.363,-176.757,8.279,148.679
C09916=1163.169,312.026,-73.395,-176.754,8.282,148.679
C09917=1163.164,312.274,-73.426,-176.752,8.286,148.679
C09918=1163.161,312.522,-73.457,-176.749,8.288,148.679
C09919=1163.156,312.770,-73.488,-176.747,8.292,148.679
C09920=1163.152,313.018,-73.520,-176.745,8.295,148.679
C09921=1163.148,313.266,-73.551,-176.742,8.298,148.679
C09922=1163.143,313.543,-73.586,-176.739,8.302,148.679
C09923=1163.138,313.821,-73.622,-176.736,8.306,148.680
C09924=1163.133,314.098,-73.657,-176.734,8.309,148.680
C09925=1163.128,314.375,-73.691,-176.730,8.313,148.680
C09926=1163.125,314.623,-73.723,-176.728,8.316,148.680
C09927=1163.121,314.871,-73.755,-176.726,8.320,148.680
C09928=1163.116,315.119,-73.786,-176.723,8.323,148.680
C09929=1163.113,315.367,-73.818,-176.721,8.326,148.680
C09930=1163.108,315.614,-73.849,-176.717,8.330,148.680
C09931=1163.104,315.863,-73.880,-176.715,8.333,148.680
C09932=1163.100,316.110,-73.912,-176.713,8.336,148.681
C09933=1163.095,316.359,-73.944,-176.710,8.339,148.681
C09934=1163.092,316.607,-73.976,-176.708,8.342,148.681
C09935=1163.087,316.855,-74.007,-176.705,8.345,148.681
C09936=1163.083,317.103,-74.039,-176.702,8.350,148.681
C09937=1163.079,317.350,-74.070,-176.700,8.353,148.681
C09938=1163.075,317.598,-74.102,-176.697,8.356,148.681
C09939=1163.071,317.847,-74.134,-176.695,8.359,148.681
C09940=1163.066,318.094,-74.165,-176.692,8.362,148.682
C09941=1163.063,318.343,-74.197,-176.690,8.365,148.682
C09942=1163.058,318.590,-74.229,-176.687,8.369,148.682
C09943=1163.054,318.838,-74.261,-176.684,8.372,148.682
C09944=1163.050,319.086,-74.293,-176.682,8.376,148.682
C09945=1163.046,319.334,-74.324,-176.679,8.379,148.682
C09946=1163.042,319.582,-74.356,-176.677,8.382,148.682
C09947=1163.038,319.830,-74.389,-176.674,8.385,148.682
C09948=1163.033,320.078,-74.419,-176.672,8.389,148.683
C09949=1163.029,320.326,-74.451,-176.669,8.392,148.683
C09950=1163.026,320.574,-74.483,-176.666,8.396,148.683
C09951=1163.021,320.822,-74.515,-176.664,8.399,148.683
C09952=1163.017,321.070,-74.547,-176.661,8.402,148.683
C09953=1163.013,321.318,-74.579,-176.659,8.405,148.683
C09954=1163.008,321.565,-74.611,-176.657,8.408,148.683
C09955=1163.005,321.813,-74.643,-176.654,8.413,148.684
C09956=1163.001,322.061,-74.675,-176.651,8.416,148.684
C09957=1162.996,322.310,-74.707,-176.649,8.419,148.684
C09958=1162.992,322.557,-74.739,-176.647,8.422,148.684
C09959=1162.988,322.805,-74.772,-176.644,8.425,148.684
C09960=1162.984,323.053,-74.804,-176.641,8.429,148.684
C09961=1162.980,323.300,-74.835,-176.639,8.433,148.684
C09962=1162.975,323.549,-74.867,-176.636,8.435,148.684
C09963=1162.972,323.797,-74.899,-176.634,8.439,148.685
C09964=1162.967,324.045,-74.932,-176.631,8.442,148.685
C09965=1162.963,324.292,-74.963,-176.628,8.446,148.685
C09966=1162.960,324.540,-74.996,-176.626,8.449,148.685
C09967=1162.955,324.788,-75.028,-176.623,8.452,148.685
C09968=1162.951,325.036,-75.060,-176.621,8.456,148.685
C09969=1162.947,325.284,-75.092,-176.618,8.459,148.685
C09970=1162.943,325.532,-75.124,-176.616,8.463,148.686
C09971=1162.939,325.780,-75.157,-176.613,8.466,148.686
C09972=1162.935,326.028,-75.189,-176.611,8.469,148.686
C09973=1162.930,326.276,-75.221,-176.608,8.472,148.686
C09974=1162.926,326.523,-75.254,-176.606,8.476,148.686
C09975=1162.922,326.771,-75.286,-176.603,8.480,148.687
C09976=1162.918,327.019,-75.318,-176.601,8.483,148.687
C09977=1162.914,327.267,-75.350,-176.598,8.486,148.687
C09978=1162.910,327.515,-75.383,-176.596,8.489,148.687
C09979=1162.905,327.762,-75.415,-176.593,8.493,148.687
C09980=1162.901,328.010,-75.448,-176.590,8.497,148.687
C09981=1162.898,328.258,-75.480,-176.588,8.500,148.688
C09982=1162.893,328.507,-75.512,-176.585,8.503,148.688
C09983=1162.890,328.754,-75.545,-176.583,8.506,148.688
C09984=1162.885,329.002,-75.577,-176.581,8.510,148.688
C09985=1162.881,329.250,-75.611,-176.578,8.514,148.688
C09986=1162.877,329.497,-75.642,-176.575,8.517,148.688
C09987=1162.873,329.745,-75.675,-176.573,8.520,148.688
C09988=1162.869,329.993,-75.707,-176.571,8.523,148.689
C09989=1162.865,330.241,-75.740,-176.568,8.527,148.689
C09990=1162.860,330.489,-75.773,-176.565,8.531,148.689
C09991=1162.857,330.737,-75.805,-176.563,8.534,148.689
C09992=1162.853,330.985,-75.838,-176.560,8.537,148.689
C09993=1162.848,331.232,-75.870,-176.558,8.541,148.689
C09994=1162.844,331.480,-75.902,-176.555,8.544,148.690
C09995=1162.840,331.728,-75.935,-176.553,8.548,148.690
C09996=1162.835,331.976,-75.968,-176.551,8.551,148.690
//INST
///DATE 2021/06/25 14:30
///ATTR SC,RW,RJ
////FRAME ROBOT
///GROUP1 RB1
NOP
MOVL C00000 V=800.0 PL=0
MOVL C00001 V=800.0 PL=0
MOVL C00002 V=800.0 PL=0
MOVL C00003 V=800.0 PL=0
MOVL C00004 V=800.0 PL=0
MOVL C00005 V=800.0 PL=0
MOVL C00006 V=800.0 PL=0
MOVL C00007 V=800.0 PL=0
MOVL C00008 V=800.0 PL=0
MOVL C00009 V=800.0 PL=0
MOVL C00010 V=800.0 PL=0
MOVL C00011 V=800.0 PL=0
MOVL C00012 V=800.0 PL=0
MOVL C00013 V=800.0 PL=0
MOVL C00014 V=800.0 PL=0
MOVL C00015 V=800.0 PL=0
MOVL C00016 V=800.0 PL=0
MOVL C00017 V=800.0 PL=0
MOVL C00018 V=800.0 PL=0
MOVL C00019 V=800.0 PL=0
MOVL C00020 V=800.0 PL=0
MOVL C00021 V=800.0 PL=0
MOVL C00022 V=800.0 PL=0
MOVL C00023 V=800.0 PL=0
MOVL C00024 V=800.0 PL=0
MOVL C00025 V=800.0 PL=0
MOVL C00026 V=800.0 PL=0
MOVL C00027 V=800.0 PL=0
MOVL C00028 V=800.0 PL=0
MOVL C00029 V=800.0 PL=0
MOVL C00030 V=800.0 PL=0
MOVL C00031 V=800.0 PL=0
MOVL C00032 V=800.0 PL=0
MOVL C00033 V=800.0 PL=0
MOVL C00034 V=800.0 PL=0
MOVL C00035 V=800.0 PL=0
MOVL C00036 V=800.0 PL=0
MOVL C00037 V=800.0 PL=0
MOVL C00038 V=800.0 PL=0
MOVL C00039 V=800.0 PL=0
MOVL C00040 V=800.0 PL=0
MOVL C00041 V=800.0 PL=0
MOVL C00042 V=800.0 PL=0
MOVL C00043 V=800.0 PL=0
MOVL C00044 V=800.0 PL=0
MOVL C00045 V=800.0 PL=0
MOVL C00046 V=800.0 PL=0
MOVL C00047 V=800.0 PL=0
MOVL C00048 V=800.0 PL=0
MOVL C00049 V=800.0 PL=0
MOVL C00050 V=800.0 PL=0
MOVL C00051 V=800.0 PL=0
MOVL C00052 V=800.0 PL=0
MOVL C00053 V=800.0 PL=0
MOVL C00054 V=800.0 PL=0
MOVL C00055 V=800.0 PL=0
MOVL C00056 V=800.0 PL=0
MOVL C00057 V=800.0 PL=0
MOVL C00058 V=800.0 PL=0
MOVL C00059 V=800.0 PL=0
MOVL C00060 V=800.0 PL=0
MOVL C00061 V=800.0 PL=0
MOVL C00062 V=800.0 PL=0
MOVL C00063 V=800.0 PL=0
MOVL C00064 V=800.0 PL=0
MOVL C00065 V=800.0 PL=0
MOVL C00066 V=800.0 PL=0
MOVL C00067 V=800.0 PL=0
MOVL C00068 V=800.0 PL=0
MOVL C00069 V=800.0 PL=0
MOVL C00070 V=800.0 PL=0
MOVL C00071 V=800.0 PL=0
MOVL C00072 V=800.0 PL=0
MOVL C00073 V=800.0 PL=0
MOVL C00074 V=800.0 PL=0
MOVL C00075 V=800.0 PL=0
MOVL C00076 V=800.0 PL=0
MOVL C00077 V=800.0 PL=0
MOVL C00078 V=800.0 PL=0
MOVL C00079 V=800.0 PL=0
MOVL C00080 V=800.0 PL=0
MOVL C00081 V=800.0 PL=0
MOVL C00082 V=800.0 PL=0
MOVL C00083 V=800.0 PL=0
MOVL C00084 V=800.0 PL=0
MOVL C00085 V=800.0 PL=0
MOVL C00086 V=800.0 PL=0
MOVL C00087 V=800.0 PL=0
MOVL C00088 V=800.0 PL=0
MOVL C00089 V=800.0 PL=0
MOVL C00090 V=800.0 PL=0
MOVL C00091 V=800.0 PL=0
MOVL C00092 V=800.0 PL=0
MOVL C00093 V=800.0 PL=0
MOVL C00094 V=800.0 PL=0
MOVL C00095 V=800.0 PL=0
MOVL C00096 V=800.0 PL=0
MOVL C00097 V=800.0 PL=0
MOVL C00098 V=800.0 PL=0
MOVL C00099 V=800.0 PL=0
MOVL C00100 V=800.0 PL=0
MOVL C00101 V=800.0 PL=0
MOVL C00102 V=800.0 PL=0
MOVL C00103 V=800.0 PL=0
MOVL C00104 V=800.0 PL=0
MOVL C00105 V=800.0 PL=0
MOVL C00106 V=800.0 PL=0
MOVL C00107 V=800.0 PL=0
MOVL C00108 V=800.0 PL=0
MOVL C00109 V=800.0 PL=0
MOVL C00110 V=800.0 PL=0
MOVL C00111 V=800.0 PL=0
MOVL C00112 V=800.0 PL=0
MOVL C00113 V=800.0 PL=0
MOVL C00114 V=800.0 PL=0
MOVL C00115 V=800.0 PL=0
MOVL C00116 V=800.0 PL=0
MOVL C00117 V=800.0 PL=0
MOVL C00118 V=800.0 PL=0
MOVL C00119 V=800.0 PL=0
MOVL C00120 V=800.0 PL=0
MOVL C00121 V=800.0 PL=0
MOVL C00122 V=800.0 PL=0
MOVL C00123 V=800.0 PL=0
MOVL C00124 V=800.0 PL=0
MOVL C00125 V=800.0 PL=0
MOVL C00126 V=800.0 PL=0
MOVL C00127 V=800.0 PL=0
MOVL C00128 V=800.0 PL=0
MOVL C00129 V=800.0 PL=0
MOVL C00130 V=800.0 PL=0
MOVL C00131 V=800.0 PL=0
MOVL C00132 V=800.0 PL=0
MOVL C00133 V=800.0 PL=0
MOVL C00134 V=800.0 PL=0
MOVL C00135 V=800.0 PL=0
MOVL C00136 V=800.0 PL=0
MOVL C00137 V=800.0 PL=0
MOVL C00138 V=800.0 PL=0
MOVL C00139 V=800.0 PL=0
MOVL C00140 V=800.0 PL=0
MOVL C00141 V=800.0 PL=0
MOVL C00142 V=800.0 PL=0
MOVL C00143 V=800.0 PL=0
MOVL C00144 V=800.0 PL=0
MOVL C00145 V=800.0 PL=0
MOVL C00146 V=800.0 PL=0
MOVL C00147 V=800.0 PL=0
MOVL C00148 V=800.0 PL=0
MOVL C00149 V=800.0 PL=0
MOVL C00150 V=800.0 PL=0
MOVL C00151 V=800.0 PL=0
MOVL C00152 V=800.0 PL=0
MOVL C00153 V=800.0 PL=0
MOVL C00154 V=800.0 PL=0
MOVL C00155 V=800.0 PL=0
MOVL C00156 V=800.0 PL=0
MOVL C00157 V=800.0 PL=0
MOVL C00158 V=800.0 PL=0
MOVL C00159 V=800.0 PL=0
MOVL C00160 V=800.0 PL=0
MOVL C00161 V=800.0 PL=0
MOVL C00162 V=800.0 PL=0
MOVL C00163 V=800.0 PL=0
MOVL C00164 V=800.0 PL=0
MOVL C00165 V=800.0 PL=0
MOVL C00166 V=800.0 PL=0
MOVL C00167 V=800.0 PL=0
MOVL C00168 V=800.0 PL=0
MOVL C00169 V=800.0 PL=0
MOVL C00170 V=800.0 PL=0
MOVL C00171 V=800.0 PL=0
MOVL C00172 V=800.0 PL=0
MOVL C00173 V=800.0 PL=0
MOVL C00174 V=800.0 PL=0
MOVL C00175 V=800.0 PL=0
MOVL C00176 V=800.0 PL=0
MOVL C00177 V=800.0 PL=0
MOVL C00178 V=800.0 PL=0
MOVL C00179 V=800.0 PL=0
MOVL C00180 V=800.0 PL=0
MOVL C00181 V=800.0 PL=0
MOVL C00182 V=800.0 PL=0
MOVL C00183 V=800.0 PL=0
MOVL C00184 V=800.0 PL=0
MOVL C00185 V=800.0 PL=0
MOVL C00186 V=800.0 PL=0
MOVL C00187 V=800.0 PL=0
MOVL C00188 V=800.0 PL=0
MOVL C00189 V=800.0 PL=0
MOVL C00190 V=800.0 PL=0
MOVL C00191 V=800.0 PL=0
MOVL C00192 V=800.0 PL=0
MOVL C00193 V=800.0 PL=0
MOVL C00194 V=800.0 PL=0
MOVL C00195 V=800.0 PL=0
MOVL C00196 V=800.0 PL=0
MOVL C00197 V=800.0 PL=0
MOVL C00198 V=800.0 PL=0
MOVL C00199 V=800.0 PL=0
MOVL C00200 V=800.0 PL=0
MOVL C00201 V=800.0 PL=0
MOVL C00202 V=800.0 PL=0
MOVL C00203 V=800.0 PL=0
MOVL C00204 V=800.0 PL=0
MOVL C00205 V=800.0 PL=0
MOVL C00206 V=800.0 PL=0
MOVL C00207 V=800.0 PL=0
MOVL C00208 V=800.0 PL=0
MOVL C00209 V=800.0 PL=0
MOVL C00210 V=800.0 PL=0
MOVL C00211 V=800.0 PL=0
MOVL C00212 V=800.0 PL=0
MOVL C00213 V=800.0 PL=0
MOVL C00214 V=800.0 PL=0
MOVL C00215 V=800.0 PL=0
MOVL C00216 V=800.0 PL=0
MOVL C00217 V=800.0 PL=0
MOVL C00218 V=800.0 PL=0
MOVL C00219 V=800.0 PL=0
MOVL C00220 V=800.0 PL=0
MOVL C00221 V=800.0 PL=0
MOVL C00222 V=800.0 PL=0
MOVL C00223 V=800.0 PL=0
MOVL C00224 V=800.0 PL=0
MOVL C00225 V=800.0 PL=0
MOVL C00226 V=800.0 PL=0
MOVL C00227 V=800.0 PL=0
MOVL C00228 V=800.0 PL=0
MOVL C00229 V=800.0 PL=0
MOVL C00230 V=800.0 PL=0
MOVL C00231 V=800.0 PL=0
MOVL C00232 V=800.0 PL=0
MOVL C00233 V=800.0 PL=0
MOVL C00234 V=800.0 PL=0
MOVL C00235 V=800.0 PL=0
MOVL C00236 V=800.0 PL=0
MOVL C00237 V=800.0 PL=0
MOVL C00238 V=800.0 PL=0
MOVL C00239 V=800.0 PL=0
MOVL C00240 V=800.0 PL=0
MOVL C00241 V=800.0 PL=0
MOVL C00242 V=800.0 PL=0
MOVL C00243 V=800.0 PL=0
MOVL C00244 V=800.0 PL=0
MOVL C00245 V=800.0 PL=0
MOVL C00246 V=800.0 PL=0
MOVL C00247 V=800.0 PL=0
MOVL C00248 V=800.0 PL=0
MOVL C00249 V=800.0 PL=0
MOVL C00250 V=800.0 PL=0
MOVL C00251 V=800.0 PL=0
MOVL C00252 V=800.0 PL=0
MOVL C00253 V=800.0 PL=0
MOVL C00254 V=800.0 PL=0
MOVL C00255 V=800.0 PL=0
MOVL C00256 V=800.0 PL=0
MOVL C00257 V=800.0 PL=0
MOVL C00258 V=800.0 PL=0
MOVL C00259 V=800.0 PL=0
MOVL C00260 V=800.0 PL=0
MOVL C00261 V=800.0 PL=0
MOVL C00262 V=800.0 PL=0
MOVL C00263 V=800.0 PL=0
MOVL C00264 V=800.0 PL=0
MOVL C00265 V=800.0 PL=0
MOVL C00266 V=800.0 PL=0
MOVL C00267 V=800.0 PL=0
MOVL C00268 V=800.0 PL=0
MOVL C00269 V=800.0 PL=0
MOVL C00270 V=800.0 PL=0
MOVL C00271 V=800.0 PL=0
MOVL C00272 V=800.0 PL=0
MOVL C00273 V=800.0 PL=0
MOVL C00274 V=800.0 PL=0
MOVL C00275 V=800.0 PL=0
MOVL C00276 V=800.0 PL=0
MOVL C00277 V=800.0 PL=0
MOVL C00278 V=800.0 PL=0
MOVL C00279 V=800.0 PL=0
MOVL C00280 V=800.0 PL=0
MOVL C00281 V=800.0 PL=0
MOVL C00282 V=800.0 PL=0
MOVL C00283 V=800.0 PL=0
MOVL C00284 V=800.0 PL=0
MOVL C00285 V=800.0 PL=0
MOVL C00286 V=800.0 PL=0
MOVL C00287 V=800.0 PL=0
MOVL C00288 V=800.0 PL=0
MOVL C00289 V=800.0 PL=0
MOVL C00290 V=800.0 PL=0
MOVL C00291 V=800.0 PL=0
MOVL C00292 V=800.0 PL=0
MOVL C00293 V=800.0 PL=0
MOVL C00294 V=800.0 PL=0
MOVL C00295 V=800.0 PL=0
MOVL C00296 V=800.0 PL=0
MOVL C00297 V=800.0 PL=0
MOVL C00298 V=800.0 PL=0
MOVL C00299 V=800.0 PL=0
MOVL C00300 V=800.0 PL=0
MOVL C00301 V=800.0 PL=0
MOVL C00302 V=800.0 PL=0
MOVL C00303 V=800.0 PL=0
MOVL C00304 V=800.0 PL=0
MOVL C00305 V=800.0 PL=0
MOVL C00306 V=800.0 PL=0
MOVL C00307 V=800.0 PL=0
MOVL C00308 V=800.0 PL=0
MOVL C00309 V=800.0 PL=0
MOVL C00310 V=800.0 PL=0
MOVL C00311 V=800.0 PL=0
MOVL C00312 V=800.0 PL=0
MOVL C00313 V=800.0 PL=0
MOVL C00314 V=800.0 PL=0
MOVL C00315 V=800.0 PL=0
MOVL C00316 V=800.0 PL=0
MOVL C00317 V=800.0 PL=0
MOVL C00318 V=800.0 PL=0
MOVL C00319 V=800.0 PL=0
MOVL C00320 V=800.0 PL=0
MOVL C00321 V=800.0 PL=0
MOVL C00322 V=800.0 PL=0
MOVL C00323 V=800.0 PL=0
MOVL C00324 V=800.0 PL=0
MOVL C00325 V=800.0 PL=0
MOVL C00326 V=800.0 PL=0
MOVL C00327 V=800.0 PL=0
MOVL C00328 V=800.0 PL=0
MOVL C00329 V=800.0 PL=0
MOVL C00330 V=800.0 PL=0
MOVL C00331 V=800.0 PL=0
MOVL C00332 V=800.0 PL=0
MOVL C00333 V=800.0 PL=0
MOVL C00334 V=800.0 PL=0
MOVL C00335 V=800.0 PL=0
MOVL C00336 V=800.0 PL=0
MOVL C00337 V=800.0 PL=0
MOVL C00338 V=800.0 PL=0
MOVL C00339 V=800.0 PL=0
MOVL C00340 V=800.0 PL=0
MOVL C00341 V=800.0 PL=0
MOVL C00342 V=800.0 PL=0
MOVL C00343 V=800.0 PL=0
MOVL C00344 V=800.0 PL=0
MOVL C00345 V=800.0 PL=0
MOVL C00346 V=800.0 PL=0
MOVL C00347 V=800.0 PL=0
MOVL C00348 V=800.0 PL=0
MOVL C00349 V=800.0 PL=0
MOVL C00350 V=800.0 PL=0
MOVL C00351 V=800.0 PL=0
MOVL C00352 V=800.0 PL=0
MOVL C00353 V=800.0 PL=0
MOVL C00354 V=800.0 PL=0
MOVL C00355 V=800.0 PL=0
MOVL C00356 V=800.0 PL=0
MOVL C00357 V=800.0 PL=0
MOVL C00358 V=800.0 PL=0
MOVL C00359 V=800.0 PL=0
MOVL C00360 V=800.0 PL=0
MOVL C00361 V=800.0 PL=0
MOVL C00362 V=800.0 PL=0
MOVL C00363 V=800.0 PL=0
MOVL C00364 V=800.0 PL=0
MOVL C00365 V=800.0 PL=0
MOVL C00366 V=800.0 PL=0
MOVL C00367 V=800.0 PL=0
MOVL C00368 V=800.0 PL=0
MOVL C00369 V=800.0 PL=0
MOVL C00370 V=800.0 PL=0
MOVL C00371 V=800.0 PL=0
MOVL C00372 V=800.0 PL=0
MOVL C00373 V=800.0 PL=0
MOVL C00374 V=800.0 PL=0
MOVL C00375 V=800.0 PL=0
MOVL C00376 V=800.0 PL=0
MOVL C00377 V=800.0 PL=0
MOVL C00378 V=800.0 PL=0
MOVL C00379 V=800.0 PL=0
MOVL C00380 V=800.0 PL=0
MOVL C00381 V=800.0 PL=0
MOVL C00382 V=800.0 PL=0
MOVL C00383 V=800.0 PL=0
MOVL C00384 V=800.0 PL=0
MOVL C00385 V=800.0 PL=0
MOVL C00386 V=800.0 PL=0
MOVL C00387 V=800.0 PL=0
MOVL C00388 V=800.0 PL=0
MOVL C00389 V=800.0 PL=0
MOVL C00390 V=800.0 PL=0
MOVL C00391 V=800.0 PL=0
MOVL C00392 V=800.0 PL=0
MOVL C00393 V=800.0 PL=0
MOVL C00394 V=800.0 PL=0
MOVL C00395 V=800.0 PL=0
MOVL C00396 V=800.0 PL=0
MOVL C00397 V=800.0 PL=0
MOVL C00398 V=800.0 PL=0
MOVL C00399 V=800.0 PL=0
MOVL C00400 V=800.0 PL=0
MOVL C00401 V=800.0 PL=0
MOVL C00402 V=800.0 PL=0
MOVL C00403 V=800.0 PL=0
MOVL C00404 V=800.0 PL=0
MOVL C00405 V=800.0 PL=0
MOVL C00406 V=800.0 PL=0
MOVL C00407 V=800.0 PL=0
MOVL C00408 V=800.0 PL=0
MOVL C00409 V=800.0 PL=0
MOVL C00410 V=800.0 PL=0
MOVL C00411 V=800.0 PL=0
MOVL C00412 V=800.0 PL=0
MOVL C00413 V=800.0 PL=0
MOVL C00414 V=800.0 PL=0
MOVL C00415 V=800.0 PL=0
MOVL C00416 V=800.0 PL=0
MOVL C00417 V=800.0 PL=0
MOVL C00418 V=800.0 PL=0
MOVL C00419 V=800.0 PL=0
MOVL C00420 V=800.0 PL=0
MOVL C00421 V=800.0 PL=0
MOVL C00422 V=800.0 PL=0
MOVL C00423 V=800.0 PL=0
MOVL C00424 V=800.0 PL=0
MOVL C00425 V=800.0 PL=0
MOVL C00426 V=800.0 PL=0
MOVL C00427 V=800.0 PL=0
MOVL C00428 V=800.0 PL=0
MOVL C00429 V=800.0 PL=0
MOVL C00430 V=800.0 PL=0
MOVL C00431 V=800.0 PL=0
MOVL C00432 V=800.0 PL=0
MOVL C00433 V=800.0 PL=0
MOVL C00434 V=800.0 PL=0
MOVL C00435 V=800.0 PL=0
MOVL C00436 V=800.0 PL=0
MOVL C00437 V=800.0 PL=0
MOVL C00438 V=800.0 PL=0
MOVL C00439 V=800.0 PL=0
MOVL C00440 V=800.0 PL=0
MOVL C00441 V=800.0 PL=0
MOVL C00442 V=800.0 PL=0
MOVL C00443 V=800.0 PL=0
MOVL C00444 V=800.0 PL=0
MOVL C00445 V=800.0 PL=0
MOVL C00446 V=800.0 PL=0
MOVL C00447 V=800.0 PL=0
MOVL C00448 V=800.0 PL=0
MOVL C00449 V=800.0 PL=0
MOVL C00450 V=800.0 PL=0
MOVL C00451 V=800.0 PL=0
MOVL C00452 V=800.0 PL=0
MOVL C00453 V=800.0 PL=0
MOVL C00454 V=800.0 PL=0
MOVL C00455 V=800.0 PL=0
MOVL C00456 V=800.0 PL=0
MOVL C00457 V=800.0 PL=0
MOVL C00458 V=800.0 PL=0
MOVL C00459 V=800.0 PL=0
MOVL C00460 V=800.0 PL=0
MOVL C00461 V=800.0 PL=0
MOVL C00462 V=800.0 PL=0
MOVL C00463 V=800.0 PL=0
MOVL C00464 V=800.0 PL=0
MOVL C00465 V=800.0 PL=0
MOVL C00466 V=800.0 PL=0
MOVL C00467 V=800.0 PL=0
MOVL C00468 V=800.0 PL=0
MOVL C00469 V=800.0 PL=0
MOVL C00470 V=800.0 PL=0
MOVL C00471 V=800.0 PL=0
MOVL C00472 V=800.0 PL=0
MOVL C00473 V=800.0 PL=0
MOVL C00474 V=800.0 PL=0
MOVL C00475 V=800.0 PL=0
MOVL C00476 V=800.0 PL=0
MOVL C00477 V=800.0 PL=0
MOVL C00478 V=800.0 PL=0
MOVL C00479 V=800.0 PL=0
MOVL C00480 V=800.0 PL=0
MOVL C00481 V=800.0 PL=0
MOVL C00482 V=800.0 PL=0
MOVL C00483 V=800.0 PL=0
MOVL C00484 V=800.0 PL=0
MOVL C00485 V=800.0 PL=0
MOVL C00486 V=800.0 PL=0
MOVL C00487 V=800.0 PL=0
MOVL C00488 V=800.0 PL=0
MOVL C00489 V=800.0 PL=0
MOVL C00490 V=800.0 PL=0
MOVL C00491 V=800.0 PL=0
MOVL C00492 V=800.0 PL=0
MOVL C00493 V=800.0 PL=0
MOVL C00494 V=800.0 PL=0
MOVL C00495 V=800.0 PL=0
MOVL C00496 V=800.0 PL=0
MOVL C00497 V=800.0 PL=0
MOVL C00498 V=800.0 PL=0
MOVL C00499 V=800.0 PL=0
MOVL C00500 V=800.0 PL=0
MOVL C00501 V=800.0 PL=0
MOVL C00502 V=800.0 PL=0
MOVL C00503 V=800.0 PL=0
MOVL C00504 V=800.0 PL=0
MOVL C00505 V=800.0 PL=0
MOVL C00506 V=800.0 PL=0
MOVL C00507 V=800.0 PL=0
MOVL C00508 V=800.0 PL=0
MOVL C00509 V=800.0 PL=0
MOVL C00510 V=800.0 PL=0
MOVL C00511 V=800.0 PL=0
MOVL C00512 V=800.0 PL=0
MOVL C00513 V=800.0 PL=0
MOVL C00514 V=800.0 PL=0
MOVL C00515 V=800.0 PL=0
MOVL C00516 V=800.0 PL=0
MOVL C00517 V=800.0 PL=0
MOVL C00518 V=800.0 PL=0
MOVL C00519 V=800.0 PL=0
MOVL C00520 V=800.0 PL=0
MOVL C00521 V=800.0 PL=0
MOVL C00522 V=800.0 PL=0
MOVL C00523 V=800.0 PL=0
MOVL C00524 V=800.0 PL=0
MOVL C00525 V=800.0 PL=0
MOVL C00526 V=800.0 PL=0
MOVL C00527 V=800.0 PL=0
MOVL C00528 V=800.0 PL=0
MOVL C00529 V=800.0 PL=0
MOVL C00530 V=800.0 PL=0
MOVL C00531 V=800.0 PL=0
MOVL C00532 V=800.0 PL=0
MOVL C00533 V=800.0 PL=0
MOVL C00534 V=800.0 PL=0
MOVL C00535 V=800.0 PL=0
MOVL C00536 V=800.0 PL=0
MOVL C00537 V=800.0 PL=0
MOVL C00538 V=800.0 PL=0
MOVL C00539 V=800.0 PL=0
MOVL C00540 V=800.0 PL=0
MOVL C00541 V=800.0 PL=0
MOVL C00542 V=800.0 PL=0
MOVL C00543 V=800.0 PL=0
MOVL C00544 V=800.0 PL=0
MOVL C00545 V=800.0 PL=0
MOVL C00546 V=800.0 PL=0
MOVL C00547 V=800.0 PL=0
MOVL C00548 V=800.0 PL=0
MOVL C00549 V=800.0 PL=0
MOVL C00550 V=800.0 PL=0
MOVL C00551 V=800.0 PL=0
MOVL C00552 V=800.0 PL=0
MOVL C00553 V=800.0 PL=0
MOVL C00554 V=800.0 PL=0
MOVL C00555 V=800.0 PL=0
MOVL C00556 V=800.0 PL=0
MOVL C00557 V=800.0 PL=0
MOVL C00558 V=800.0 PL=0
MOVL C00559 V=800.0 PL=0
MOVL C00560 V=800.0 PL=0
MOVL C00561 V=800.0 PL=0
MOVL C00562 V=800.0 PL=0
MOVL C00563 V=800.0 PL=0
MOVL C00564 V=800.0 PL=0
MOVL C00565 V=800.0 PL=0
MOVL C00566 V=800.0 PL=0
MOVL C00567 V=800.0 PL=0
MOVL C00568 V=800.0 PL=0
MOVL C00569 V=800.0 PL=0
MOVL C00570 V=800.0 PL=0
MOVL C00571 V=800.0 PL=0
MOVL C00572 V=800.0 PL=0
MOVL C00573 V=800.0 PL=0
MOVL C00574 V=800.0 PL=0
MOVL C00575 V=800.0 PL=0
MOVL C00576 V=800.0 PL=0
MOVL C00577 V=800.0 PL=0
MOVL C00578 V=800.0 PL=0
MOVL C00579 V=800.0 PL=0
MOVL C00580 V=800.0 PL=0
MOVL C00581 V=800.0 PL=0
MOVL C00582 V=800.0 PL=0
MOVL C00583 V=800.0 PL=0
MOVL C00584 V=800.0 PL=0
MOVL C00585 V=800.0 PL=0
MOVL C00586 V=800.0 PL=0
MOVL C00587 V=800.0 PL=0
MOVL C00588 V=800.0 PL=0
MOVL C00589 V=800.0 PL=0
MOVL C00590 V=800.0 PL=0
MOVL C00591 V=800.0 PL=0
MOVL C00592 V=800.0 PL=0
MOVL C00593 V=800.0 PL=0
MOVL C00594 V=800.0 PL=0
MOVL C00595 V=800.0 PL=0
MOVL C00596 V=800.0 PL=0
MOVL C00597 V=800.0 PL=0
MOVL C00598 V=800.0 PL=0
MOVL C00599 V=800.0 PL=0
MOVL C00600 V=800.0 PL=0
MOVL C00601 V=800.0 PL=0
MOVL C00602 V=800.0 PL=0
MOVL C00603 V=800.0 PL=0
MOVL C00604 V=800.0 PL=0
MOVL C00605 V=800.0 PL=0
MOVL C00606 V=800.0 PL=0
MOVL C00607 V=800.0 PL=0
MOVL C00608 V=800.0 PL=0
MOVL C00609 V=800.0 PL=0
MOVL C00610 V=800.0 PL=0
MOVL C00611 V=800.0 PL=0
MOVL C00612 V=800.0 PL=0
MOVL C00613 V=800.0 PL=0
MOVL C00614 V=800.0 PL=0
MOVL C00615 V=800.0 PL=0
MOVL C00616 V=800.0 PL=0
MOVL C00617 V=800.0 PL=0
MOVL C00618 V=800.0 PL=0
MOVL C00619 V=800.0 PL=0
MOVL C00620 V=800.0 PL=0
MOVL C00621 V=800.0 PL=0
MOVL C00622 V=800.0 PL=0
MOVL C00623 V=800.0 PL=0
MOVL C00624 V=800.0 PL=0
MOVL C00625 V=800.0 PL=0
MOVL C00626 V=800.0 PL=0
MOVL C00627 V=800.0 PL=0
MOVL C00628 V=800.0 PL=0
MOVL C00629 V=800.0 PL=0
MOVL C00630 V=800.0 PL=0
MOVL C00631 V=800.0 PL=0
MOVL C00632 V=800.0 PL=0
MOVL C00633 V=800.0 PL=0
MOVL C00634 V=800.0 PL=0
MOVL C00635 V=800.0 PL=0
MOVL C00636 V=800.0 PL=0
MOVL C00637 V=800.0 PL=0
MOVL C00638 V=800.0 PL=0
MOVL C00639 V=800.0 PL=0
MOVL C00640 V=800.0 PL=0
MOVL C00641 V=800.0 PL=0
MOVL C00642 V=800.0 PL=0
MOVL C00643 V=800.0 PL=0
MOVL C00644 V=800.0 PL=0
MOVL C00645 V=800.0 PL=0
MOVL C00646 V=800.0 PL=0
MOVL C00647 V=800.0 PL=0
MOVL C00648 V=800.0 PL=0
MOVL C00649 V=800.0 PL=0
MOVL C00650 V=800.0 PL=0
MOVL C00651 V=800.0 PL=0
MOVL C00652 V=800.0 PL=0
MOVL C00653 V=800.0 PL=0
MOVL C00654 V=800.0 PL=0
MOVL C00655 V=800.0 PL=0
MOVL C00656 V=800.0 PL=0
MOVL C00657 V=800.0 PL=0
MOVL C00658 V=800.0 PL=0
MOVL C00659 V=800.0 PL=0
MOVL C00660 V=800.0 PL=0
MOVL C00661 V=800.0 PL=0
MOVL C00662 V=800.0 PL=0
MOVL C00663 V=800.0 PL=0
MOVL C00664 V=800.0 PL=0
MOVL C00665 V=800.0 PL=0
MOVL C00666 V=800.0 PL=0
MOVL C00667 V=800.0 PL=0
MOVL C00668 V=800.0 PL=0
MOVL C00669 V=800.0 PL=0
MOVL C00670 V=800.0 PL=0
MOVL C00671 V=800.0 PL=0
MOVL C00672 V=800.0 PL=0
MOVL C00673 V=800.0 PL=0
MOVL C00674 V=800.0 PL=0
MOVL C00675 V=800.0 PL=0
MOVL C00676 V=800.0 PL=0
MOVL C00677 V=800.0 PL=0
MOVL C00678 V=800.0 PL=0
MOVL C00679 V=800.0 PL=0
MOVL C00680 V=800.0 PL=0
MOVL C00681 V=800.0 PL=0
MOVL C00682 V=800.0 PL=0
MOVL C00683 V=800.0 PL=0
MOVL C00684 V=800.0 PL=0
MOVL C00685 V=800.0 PL=0
MOVL C00686 V=800.0 PL=0
MOVL C00687 V=800.0 PL=0
MOVL C00688 V=800.0 PL=0
MOVL C00689 V=800.0 PL=0
MOVL C00690 V=800.0 PL=0
MOVL C00691 V=800.0 PL=0
MOVL C00692 V=800.0 PL=0
MOVL C00693 V=800.0 PL=0
MOVL C00694 V=800.0 PL=0
MOVL C00695 V=800.0 PL=0
MOVL C00696 V=800.0 PL=0
MOVL C00697 V=800.0 PL=0
MOVL C00698 V=800.0 PL=0
MOVL C00699 V=800.0 PL=0
MOVL C00700 V=800.0 PL=0
MOVL C00701 V=800.0 PL=0
MOVL C00702 V=800.0 PL=0
MOVL C00703 V=800.0 PL=0
MOVL C00704 V=800.0 PL=0
MOVL C00705 V=800.0 PL=0
MOVL C00706 V=800.0 PL=0
MOVL C00707 V=800.0 PL=0
MOVL C00708 V=800.0 PL=0
MOVL C00709 V=800.0 PL=0
MOVL C00710 V=800.0 PL=0
MOVL C00711 V=800.0 PL=0
MOVL C00712 V=800.0 PL=0
MOVL C00713 V=800.0 PL=0
MOVL C00714 V=800.0 PL=0
MOVL C00715 V=800.0 PL=0
MOVL C00716 V=800.0 PL=0
MOVL C00717 V=800.0 PL=0
MOVL C00718 V=800.0 PL=0
MOVL C00719 V=800.0 PL=0
MOVL C00720 V=800.0 PL=0
MOVL C00721 V=800.0 PL=0
MOVL C00722 V=800.0 PL=0
MOVL C00723 V=800.0 PL=0
MOVL C00724 V=800.0 PL=0
MOVL C00725 V=800.0 PL=0
MOVL C00726 V=800.0 PL=0
MOVL C00727 V=800.0 PL=0
MOVL C00728 V=800.0 PL=0
MOVL C00729 V=800.0 PL=0
MOVL C00730 V=800.0 PL=0
MOVL C00731 V=800.0 PL=0
MOVL C00732 V=800.0 PL=0
MOVL C00733 V=800.0 PL=0
MOVL C00734 V=800.0 PL=0
MOVL C00735 V=800.0 PL=0
MOVL C00736 V=800.0 PL=0
MOVL C00737 V=800.0 PL=0
MOVL C00738 V=800.0 PL=0
MOVL C00739 V=800.0 PL=0
MOVL C00740 V=800.0 PL=0
MOVL C00741 V=800.0 PL=0
MOVL C00742 V=800.0 PL=0
MOVL C00743 V=800.0 PL=0
MOVL C00744 V=800.0 PL=0
MOVL C00745 V=800.0 PL=0
MOVL C00746 V=800.0 PL=0
MOVL C00747 V=800.0 PL=0
MOVL C00748 V=800.0 PL=0
MOVL C00749 V=800.0 PL=0
MOVL C00750 V=800.0 PL=0
MOVL C00751 V=800.0 PL=0
MOVL C00752 V=800.0 PL=0
MOVL C00753 V=800.0 PL=0
MOVL C00754 V=800.0 PL=0
MOVL C00755 V=800.0 PL=0
MOVL C00756 V=800.0 PL=0
MOVL C00757 V=800.0 PL=0
MOVL C00758 V=800.0 PL=0
MOVL C00759 V=800.0 PL=0
MOVL C00760 V=800.0 PL=0
MOVL C00761 V=800.0 PL=0
MOVL C00762 V=800.0 PL=0
MOVL C00763 V=800.0 PL=0
MOVL C00764 V=800.0 PL=0
MOVL C00765 V=800.0 PL=0
MOVL C00766 V=800.0 PL=0
MOVL C00767 V=800.0 PL=0
MOVL C00768 V=800.0 PL=0
MOVL C00769 V=800.0 PL=0
MOVL C00770 V=800.0 PL=0
MOVL C00771 V=800.0 PL=0
MOVL C00772 V=800.0 PL=0
MOVL C00773 V=800.0 PL=0
MOVL C00774 V=800.0 PL=0
MOVL C00775 V=800.0 PL=0
MOVL C00776 V=800.0 PL=0
MOVL C00777 V=800.0 PL=0
MOVL C00778 V=800.0 PL=0
MOVL C00779 V=800.0 PL=0
MOVL C00780 V=800.0 PL=0
MOVL C00781 V=800.0 PL=0
MOVL C00782 V=800.0 PL=0
MOVL C00783 V=800.0 PL=0
MOVL C00784 V=800.0 PL=0
MOVL C00785 V=800.0 PL=0
MOVL C00786 V=800.0 PL=0
MOVL C00787 V=800.0 PL=0
MOVL C00788 V=800.0 PL=0
MOVL C00789 V=800.0 PL=0
MOVL C00790 V=800.0 PL=0
MOVL C00791 V=800.0 PL=0
MOVL C00792 V=800.0 PL=0
MOVL C00793 V=800.0 PL=0
MOVL C00794 V=800.0 PL=0
MOVL C00795 V=800.0 PL=0
MOVL C00796 V=800.0 PL=0
MOVL C00797 V=800.0 PL=0
MOVL C00798 V=800.0 PL=0
MOVL C00799 V=800.0 PL=0
MOVL C00800 V=800.0 PL=0
MOVL C00801 V=800.0 PL=0
MOVL C00802 V=800.0 PL=0
MOVL C00803 V=800.0 PL=0
MOVL C00804 V=800.0 PL=0
MOVL C00805 V=800.0 PL=0
MOVL C00806 V=800.0 PL=0
MOVL C00807 V=800.0 PL=0
MOVL C00808 V=800.0 PL=0
MOVL C00809 V=800.0 PL=0
MOVL C00810 V=800.0 PL=0
MOVL C00811 V=800.0 PL=0
MOVL C00812 V=800.0 PL=0
MOVL C00813 V=800.0 PL=0
MOVL C00814 V=800.0 PL=0
MOVL C00815 V=800.0 PL=0
MOVL C00816 V=800.0 PL=0
MOVL C00817 V=800.0 PL=0
MOVL C00818 V=800.0 PL=0
MOVL C00819 V=800.0 PL=0
MOVL C00820 V=800.0 PL=0
MOVL C00821 V=800.0 PL=0
MOVL C00822 V=800.0 PL=0
MOVL C00823 V=800.0 PL=0
MOVL C00824 V=800.0 PL=0
MOVL C00825 V=800.0 PL=0
MOVL C00826 V=800.0 PL=0
MOVL C00827 V=800.0 PL=0
MOVL C00828 V=800.0 PL=0
MOVL C00829 V=800.0 PL=0
MOVL C00830 V=800.0 PL=0
MOVL C00831 V=800.0 PL=0
MOVL C00832 V=800.0 PL=0
MOVL C00833 V=800.0 PL=0
MOVL C00834 V=800.0 PL=0
MOVL C00835 V=800.0 PL=0
MOVL C00836 V=800.0 PL=0
MOVL C00837 V=800.0 PL=0
MOVL C00838 V=800.0 PL=0
MOVL C00839 V=800.0 PL=0
MOVL C00840 V=800.0 PL=0
MOVL C00841 V=800.0 PL=0
MOVL C00842 V=800.0 PL=0
MOVL C00843 V=800.0 PL=0
MOVL C00844 V=800.0 PL=0
MOVL C00845 V=800.0 PL=0
MOVL C00846 V=800.0 PL=0
MOVL C00847 V=800.0 PL=0
MOVL C00848 V=800.0 PL=0
MOVL C00849 V=800.0 PL=0
MOVL C00850 V=800.0 PL=0
MOVL C00851 V=800.0 PL=0
MOVL C00852 V=800.0 PL=0
MOVL C00853 V=800.0 PL=0
MOVL C00854 V=800.0 PL=0
MOVL C00855 V=800.0 PL=0
MOVL C00856 V=800.0 PL=0
MOVL C00857 V=800.0 PL=0
MOVL C00858 V=800.0 PL=0
MOVL C00859 V=800.0 PL=0
MOVL C00860 V=800.0 PL=0
MOVL C00861 V=800.0 PL=0
MOVL C00862 V=800.0 PL=0
MOVL C00863 V=800.0 PL=0
MOVL C00864 V=800.0 PL=0
MOVL C00865 V=800.0 PL=0
MOVL C00866 V=800.0 PL=0
MOVL C00867 V=800.0 PL=0
MOVL C00868 V=800.0 PL=0
MOVL C00869 V=800.0 PL=0
MOVL C00870 V=800.0 PL=0
MOVL C00871 V=800.0 PL=0
MOVL C00872 V=800.0 PL=0
MOVL C00873 V=800.0 PL=0
MOVL C00874 V=800.0 PL=0
MOVL C00875 V=800.0 PL=0
MOVL C00876 V=800.0 PL=0
MOVL C00877 V=800.0 PL=0
MOVL C00878 V=800.0 PL=0
MOVL C00879 V=800.0 PL=0
MOVL C00880 V=800.0 PL=0
MOVL C00881 V=800.0 PL=0
MOVL C00882 V=800.0 PL=0
MOVL C00883 V=800.0 PL=0
MOVL C00884 V=800.0 PL=0
MOVL C00885 V=800.0 PL=0
MOVL C00886 V=800.0 PL=0
MOVL C00887 V=800.0 PL=0
MOVL C00888 V=800.0 PL=0
MOVL C00889 V=800.0 PL=0
MOVL C00890 V=800.0 PL=0
MOVL C00891 V=800.0 PL=0
MOVL C00892 V=800.0 PL=0
MOVL C00893 V=800.0 PL=0
MOVL C00894 V=800.0 PL=0
MOVL C00895 V=800.0 PL=0
MOVL C00896 V=800.0 PL=0
MOVL C00897 V=800.0 PL=0
MOVL C00898 V=800.0 PL=0
MOVL C00899 V=800.0 PL=0
MOVL C00900 V=800.0 PL=0
MOVL C00901 V=800.0 PL=0
MOVL C00902 V=800.0 PL=0
MOVL C00903 V=800.0 PL=0
MOVL C00904 V=800.0 PL=0
MOVL C00905 V=800.0 PL=0
MOVL C00906 V=800.0 PL=0
MOVL C00907 V=800.0 PL=0
MOVL C00908 V=800.0 PL=0
MOVL C00909 V=800.0 PL=0
MOVL C00910 V=800.0 PL=0
MOVL C00911 V=800.0 PL=0
MOVL C00912 V=800.0 PL=0
MOVL C00913 V=800.0 PL=0
MOVL C00914 V=800.0 PL=0
MOVL C00915 V=800.0 PL=0
MOVL C00916 V=800.0 PL=0
MOVL C00917 V=800.0 PL=0
MOVL C00918 V=800.0 PL=0
MOVL C00919 V=800.0 PL=0
MOVL C00920 V=800.0 PL=0
MOVL C00921 V=800.0 PL=0
MOVL C00922 V=800.0 PL=0
MOVL C00923 V=800.0 PL=0
MOVL C00924 V=800.0 PL=0
MOVL C00925 V=800.0 PL=0
MOVL C00926 V=800.0 PL=0
MOVL C00927 V=800.0 PL=0
MOVL C00928 V=800.0 PL=0
MOVL C00929 V=800.0 PL=0
MOVL C00930 V=800.0 PL=0
MOVL C00931 V=800.0 PL=0
MOVL C00932 V=800.0 PL=0
MOVL C00933 V=800.0 PL=0
MOVL C00934 V=800.0 PL=0
MOVL C00935 V=800.0 PL=0
MOVL C00936 V=800.0 PL=0
MOVL C00937 V=800.0 PL=0
MOVL C00938 V=800.0 PL=0
MOVL C00939 V=800.0 PL=0
MOVL C00940 V=800.0 PL=0
MOVL C00941 V=800.0 PL=0
MOVL C00942 V=800.0 PL=0
MOVL C00943 V=800.0 PL=0
MOVL C00944 V=800.0 PL=0
MOVL C00945 V=800.0 PL=0
MOVL C00946 V=800.0 PL=0
MOVL C00947 V=800.0 PL=0
MOVL C00948 V=800.0 PL=0
MOVL C00949 V=800.0 PL=0
MOVL C00950 V=800.0 PL=0
MOVL C00951 V=800.0 PL=0
MOVL C00952 V=800.0 PL=0
MOVL C00953 V=800.0 PL=0
MOVL C00954 V=800.0 PL=0
MOVL C00955 V=800.0 PL=0
MOVL C00956 V=800.0 PL=0
MOVL C00957 V=800.0 PL=0
MOVL C00958 V=800.0 PL=0
MOVL C00959 V=800.0 PL=0
MOVL C00960 V=800.0 PL=0
MOVL C00961 V=800.0 PL=0
MOVL C00962 V=800.0 PL=0
MOVL C00963 V=800.0 PL=0
MOVL C00964 V=800.0 PL=0
MOVL C00965 V=800.0 PL=0
MOVL C00966 V=800.0 PL=0
MOVL C00967 V=800.0 PL=0
MOVL C00968 V=800.0 PL=0
MOVL C00969 V=800.0 PL=0
MOVL C00970 V=800.0 PL=0
MOVL C00971 V=800.0 PL=0
MOVL C00972 V=800.0 PL=0
MOVL C00973 V=800.0 PL=0
MOVL C00974 V=800.0 PL=0
MOVL C00975 V=800.0 PL=0
MOVL C00976 V=800.0 PL=0
MOVL C00977 V=800.0 PL=0
MOVL C00978 V=800.0 PL=0
MOVL C00979 V=800.0 PL=0
MOVL C00980 V=800.0 PL=0
MOVL C00981 V=800.0 PL=0
MOVL C00982 V=800.0 PL=0
MOVL C00983 V=800.0 PL=0
MOVL C00984 V=800.0 PL=0
MOVL C00985 V=800.0 PL=0
MOVL C00986 V=800.0 PL=0
MOVL C00987 V=800.0 PL=0
MOVL C00988 V=800.0 PL=0
MOVL C00989 V=800.0 PL=0
MOVL C00990 V=800.0 PL=0
MOVL C00991 V=800.0 PL=0
MOVL C00992 V=800.0 PL=0
MOVL C00993 V=800.0 PL=0
MOVL C00994 V=800.0 PL=0
MOVL C00995 V=800.0 PL=0
MOVL C00996 V=800.0 PL=0
MOVL C00997 V=800.0 PL=0
MOVL C00998 V=800.0 PL=0
MOVL C00999 V=800.0 PL=0
MOVL C01000 V=800.0 PL=0
MOVL C01001 V=800.0 PL=0
MOVL C01002 V=800.0 PL=0
MOVL C01003 V=800.0 PL=0
MOVL C01004 V=800.0 PL=0
MOVL C01005 V=800.0 PL=0
MOVL C01006 V=800.0 PL=0
MOVL C01007 V=800.0 PL=0
MOVL C01008 V=800.0 PL=0
MOVL C01009 V=800.0 PL=0
MOVL C01010 V=800.0 PL=0
MOVL C01011 V=800.0 PL=0
MOVL C01012 V=800.0 PL=0
MOVL C01013 V=800.0 PL=0
MOVL C01014 V=800.0 PL=0
MOVL C01015 V=800.0 PL=0
MOVL C01016 V=800.0 PL=0
MOVL C01017 V=800.0 PL=0
MOVL C01018 V=800.0 PL=0
MOVL C01019 V=800.0 PL=0
MOVL C01020 V=800.0 PL=0
MOVL C01021 V=800.0 PL=0
MOVL C01022 V=800.0 PL=0
MOVL C01023 V=800.0 PL=0
MOVL C01024 V=800.0 PL=0
MOVL C01025 V=800.0 PL=0
MOVL C01026 V=800.0 PL=0
MOVL C01027 V=800.0 PL=0
MOVL C01028 V=800.0 PL=0
MOVL C01029 V=800.0 PL=0
MOVL C01030 V=800.0 PL=0
MOVL C01031 V=800.0 PL=0
MOVL C01032 V=800.0 PL=0
MOVL C01033 V=800.0 PL=0
MOVL C01034 V=800.0 PL=0
MOVL C01035 V=800.0 PL=0
MOVL C01036 V=800.0 PL=0
MOVL C01037 V=800.0 PL=0
MOVL C01038 V=800.0 PL=0
MOVL C01039 V=800.0 PL=0
MOVL C01040 V=800.0 PL=0
MOVL C01041 V=800.0 PL=0
MOVL C01042 V=800.0 PL=0
MOVL C01043 V=800.0 PL=0
MOVL C01044 V=800.0 PL=0
MOVL C01045 V=800.0 PL=0
MOVL C01046 V=800.0 PL=0
MOVL C01047 V=800.0 PL=0
MOVL C01048 V=800.0 PL=0
MOVL C01049 V=800.0 PL=0
MOVL C01050 V=800.0 PL=0
MOVL C01051 V=800.0 PL=0
MOVL C01052 V=800.0 PL=0
MOVL C01053 V=800.0 PL=0
MOVL C01054 V=800.0 PL=0
MOVL C01055 V=800.0 PL=0
MOVL C01056 V=800.0 PL=0
MOVL C01057 V=800.0 PL=0
MOVL C01058 V=800.0 PL=0
MOVL C01059 V=800.0 PL=0
MOVL C01060 V=800.0 PL=0
MOVL C01061 V=800.0 PL=0
MOVL C01062 V=800.0 PL=0
MOVL C01063 V=800.0 PL=0
MOVL C01064 V=800.0 PL=0
MOVL C01065 V=800.0 PL=0
MOVL C01066 V=800.0 PL=0
MOVL C01067 V=800.0 PL=0
MOVL C01068 V=800.0 PL=0
MOVL C01069 V=800.0 PL=0
MOVL C01070 V=800.0 PL=0
MOVL C01071 V=800.0 PL=0
MOVL C01072 V=800.0 PL=0
MOVL C01073 V=800.0 PL=0
MOVL C01074 V=800.0 PL=0
MOVL C01075 V=800.0 PL=0
MOVL C01076 V=800.0 PL=0
MOVL C01077 V=800.0 PL=0
MOVL C01078 V=800.0 PL=0
MOVL C01079 V=800.0 PL=0
MOVL C01080 V=800.0 PL=0
MOVL C01081 V=800.0 PL=0
MOVL C01082 V=800.0 PL=0
MOVL C01083 V=800.0 PL=0
MOVL C01084 V=800.0 PL=0
MOVL C01085 V=800.0 PL=0
MOVL C01086 V=800.0 PL=0
MOVL C01087 V=800.0 PL=0
MOVL C01088 V=800.0 PL=0
MOVL C01089 V=800.0 PL=0
MOVL C01090 V=800.0 PL=0
MOVL C01091 V=800.0 PL=0
MOVL C01092 V=800.0 PL=0
MOVL C01093 V=800.0 PL=0
MOVL C01094 V=800.0 PL=0
MOVL C01095 V=800.0 PL=0
MOVL C01096 V=800.0 PL=0
MOVL C01097 V=800.0 PL=0
MOVL C01098 V=800.0 PL=0
MOVL C01099 V=800.0 PL=0
MOVL C01100 V=800.0 PL=0
MOVL C01101 V=800.0 PL=0
MOVL C01102 V=800.0 PL=0
MOVL C01103 V=800.0 PL=0
MOVL C01104 V=800.0 PL=0
MOVL C01105 V=800.0 PL=0
MOVL C01106 V=800.0 PL=0
MOVL C01107 V=800.0 PL=0
MOVL C01108 V=800.0 PL=0
MOVL C01109 V=800.0 PL=0
MOVL C01110 V=800.0 PL=0
MOVL C01111 V=800.0 PL=0
MOVL C01112 V=800.0 PL=0
MOVL C01113 V=800.0 PL=0
MOVL C01114 V=800.0 PL=0
MOVL C01115 V=800.0 PL=0
MOVL C01116 V=800.0 PL=0
MOVL C01117 V=800.0 PL=0
MOVL C01118 V=800.0 PL=0
MOVL C01119 V=800.0 PL=0
MOVL C01120 V=800.0 PL=0
MOVL C01121 V=800.0 PL=0
MOVL C01122 V=800.0 PL=0
MOVL C01123 V=800.0 PL=0
MOVL C01124 V=800.0 PL=0
MOVL C01125 V=800.0 PL=0
MOVL C01126 V=800.0 PL=0
MOVL C01127 V=800.0 PL=0
MOVL C01128 V=800.0 PL=0
MOVL C01129 V=800.0 PL=0
MOVL C01130 V=800.0 PL=0
MOVL C01131 V=800.0 PL=0
MOVL C01132 V=800.0 PL=0
MOVL C01133 V=800.0 PL=0
MOVL C01134 V=800.0 PL=0
MOVL C01135 V=800.0 PL=0
MOVL C01136 V=800.0 PL=0
MOVL C01137 V=800.0 PL=0
MOVL C01138 V=800.0 PL=0
MOVL C01139 V=800.0 PL=0
MOVL C01140 V=800.0 PL=0
MOVL C01141 V=800.0 PL=0
MOVL C01142 V=800.0 PL=0
MOVL C01143 V=800.0 PL=0
MOVL C01144 V=800.0 PL=0
MOVL C01145 V=800.0 PL=0
MOVL C01146 V=800.0 PL=0
MOVL C01147 V=800.0 PL=0
MOVL C01148 V=800.0 PL=0
MOVL C01149 V=800.0 PL=0
MOVL C01150 V=800.0 PL=0
MOVL C01151 V=800.0 PL=0
MOVL C01152 V=800.0 PL=0
MOVL C01153 V=800.0 PL=0
MOVL C01154 V=800.0 PL=0
MOVL C01155 V=800.0 PL=0
MOVL C01156 V=800.0 PL=0
MOVL C01157 V=800.0 PL=0
MOVL C01158 V=800.0 PL=0
MOVL C01159 V=800.0 PL=0
MOVL C01160 V=800.0 PL=0
MOVL C01161 V=800.0 PL=0
MOVL C01162 V=800.0 PL=0
MOVL C01163 V=800.0 PL=0
MOVL C01164 V=800.0 PL=0
MOVL C01165 V=800.0 PL=0
MOVL C01166 V=800.0 PL=0
MOVL C01167 V=800.0 PL=0
MOVL C01168 V=800.0 PL=0
MOVL C01169 V=800.0 PL=0
MOVL C01170 V=800.0 PL=0
MOVL C01171 V=800.0 PL=0
MOVL C01172 V=800.0 PL=0
MOVL C01173 V=800.0 PL=0
MOVL C01174 V=800.0 PL=0
MOVL C01175 V=800.0 PL=0
MOVL C01176 V=800.0 PL=0
MOVL C01177 V=800.0 PL=0
MOVL C01178 V=800.0 PL=0
MOVL C01179 V=800.0 PL=0
MOVL C01180 V=800.0 PL=0
MOVL C01181 V=800.0 PL=0
MOVL C01182 V=800.0 PL=0
MOVL C01183 V=800.0 PL=0
MOVL C01184 V=800.0 PL=0
MOVL C01185 V=800.0 PL=0
MOVL C01186 V=800.0 PL=0
MOVL C01187 V=800.0 PL=0
MOVL C01188 V=800.0 PL=0
MOVL C01189 V=800.0 PL=0
MOVL C01190 V=800.0 PL=0
MOVL C01191 V=800.0 PL=0
MOVL C01192 V=800.0 PL=0
MOVL C01193 V=800.0 PL=0
MOVL C01194 V=800.0 PL=0
MOVL C01195 V=800.0 PL=0
MOVL C01196 V=800.0 PL=0
MOVL C01197 V=800.0 PL=0
MOVL C01198 V=800.0 PL=0
MOVL C01199 V=800.0 PL=0
MOVL C01200 V=800.0 PL=0
MOVL C01201 V=800.0 PL=0
MOVL C01202 V=800.0 PL=0
MOVL C01203 V=800.0 PL=0
MOVL C01204 V=800.0 PL=0
MOVL C01205 V=800.0 PL=0
MOVL C01206 V=800.0 PL=0
MOVL C01207 V=800.0 PL=0
MOVL C01208 V=800.0 PL=0
MOVL C01209 V=800.0 PL=0
MOVL C01210 V=800.0 PL=0
MOVL C01211 V=800.0 PL=0
MOVL C01212 V=800.0 PL=0
MOVL C01213 V=800.0 PL=0
MOVL C01214 V=800.0 PL=0
MOVL C01215 V=800.0 PL=0
MOVL C01216 V=800.0 PL=0
MOVL C01217 V=800.0 PL=0
MOVL C01218 V=800.0 PL=0
MOVL C01219 V=800.0 PL=0
MOVL C01220 V=800.0 PL=0
MOVL C01221 V=800.0 PL=0
MOVL C01222 V=800.0 PL=0
MOVL C01223 V=800.0 PL=0
MOVL C01224 V=800.0 PL=0
MOVL C01225 V=800.0 PL=0
MOVL C01226 V=800.0 PL=0
MOVL C01227 V=800.0 PL=0
MOVL C01228 V=800.0 PL=0
MOVL C01229 V=800.0 PL=0
MOVL C01230 V=800.0 PL=0
MOVL C01231 V=800.0 PL=0
MOVL C01232 V=800.0 PL=0
MOVL C01233 V=800.0 PL=0
MOVL C01234 V=800.0 PL=0
MOVL C01235 V=800.0 PL=0
MOVL C01236 V=800.0 PL=0
MOVL C01237 V=800.0 PL=0
MOVL C01238 V=800.0 PL=0
MOVL C01239 V=800.0 PL=0
MOVL C01240 V=800.0 PL=0
MOVL C01241 V=800.0 PL=0
MOVL C01242 V=800.0 PL=0
MOVL C01243 V=800.0 PL=0
MOVL C01244 V=800.0 PL=0
MOVL C01245 V=800.0 PL=0
MOVL C01246 V=800.0 PL=0
MOVL C01247 V=800.0 PL=0
MOVL C01248 V=800.0 PL=0
MOVL C01249 V=800.0 PL=0
MOVL C01250 V=800.0 PL=0
MOVL C01251 V=800.0 PL=0
MOVL C01252 V=800.0 PL=0
MOVL C01253 V=800.0 PL=0
MOVL C01254 V=800.0 PL=0
MOVL C01255 V=800.0 PL=0
MOVL C01256 V=800.0 PL=0
MOVL C01257 V=800.0 PL=0
MOVL C01258 V=800.0 PL=0
MOVL C01259 V=800.0 PL=0
MOVL C01260 V=800.0 PL=0
MOVL C01261 V=800.0 PL=0
MOVL C01262 V=800.0 PL=0
MOVL C01263 V=800.0 PL=0
MOVL C01264 V=800.0 PL=0
MOVL C01265 V=800.0 PL=0
MOVL C01266 V=800.0 PL=0
MOVL C01267 V=800.0 PL=0
MOVL C01268 V=800.0 PL=0
MOVL C01269 V=800.0 PL=0
MOVL C01270 V=800.0 PL=0
MOVL C01271 V=800.0 PL=0
MOVL C01272 V=800.0 PL=0
MOVL C01273 V=800.0 PL=0
MOVL C01274 V=800.0 PL=0
MOVL C01275 V=800.0 PL=0
MOVL C01276 V=800.0 PL=0
MOVL C01277 V=800.0 PL=0
MOVL C01278 V=800.0 PL=0
MOVL C01279 V=800.0 PL=0
MOVL C01280 V=800.0 PL=0
MOVL C01281 V=800.0 PL=0
MOVL C01282 V=800.0 PL=0
MOVL C01283 V=800.0 PL=0
MOVL C01284 V=800.0 PL=0
MOVL C01285 V=800.0 PL=0
MOVL C01286 V=800.0 PL=0
MOVL C01287 V=800.0 PL=0
MOVL C01288 V=800.0 PL=0
MOVL C01289 V=800.0 PL=0
MOVL C01290 V=800.0 PL=0
MOVL C01291 V=800.0 PL=0
MOVL C01292 V=800.0 PL=0
MOVL C01293 V=800.0 PL=0
MOVL C01294 V=800.0 PL=0
MOVL C01295 V=800.0 PL=0
MOVL C01296 V=800.0 PL=0
MOVL C01297 V=800.0 PL=0
MOVL C01298 V=800.0 PL=0
MOVL C01299 V=800.0 PL=0
MOVL C01300 V=800.0 PL=0
MOVL C01301 V=800.0 PL=0
MOVL C01302 V=800.0 PL=0
MOVL C01303 V=800.0 PL=0
MOVL C01304 V=800.0 PL=0
MOVL C01305 V=800.0 PL=0
MOVL C01306 V=800.0 PL=0
MOVL C01307 V=800.0 PL=0
MOVL C01308 V=800.0 PL=0
MOVL C01309 V=800.0 PL=0
MOVL C01310 V=800.0 PL=0
MOVL C01311 V=800.0 PL=0
MOVL C01312 V=800.0 PL=0
MOVL C01313 V=800.0 PL=0
MOVL C01314 V=800.0 PL=0
MOVL C01315 V=800.0 PL=0
MOVL C01316 V=800.0 PL=0
MOVL C01317 V=800.0 PL=0
MOVL C01318 V=800.0 PL=0
MOVL C01319 V=800.0 PL=0
MOVL C01320 V=800.0 PL=0
MOVL C01321 V=800.0 PL=0
MOVL C01322 V=800.0 PL=0
MOVL C01323 V=800.0 PL=0
MOVL C01324 V=800.0 PL=0
MOVL C01325 V=800.0 PL=0
MOVL C01326 V=800.0 PL=0
MOVL C01327 V=800.0 PL=0
MOVL C01328 V=800.0 PL=0
MOVL C01329 V=800.0 PL=0
MOVL C01330 V=800.0 PL=0
MOVL C01331 V=800.0 PL=0
MOVL C01332 V=800.0 PL=0
MOVL C01333 V=800.0 PL=0
MOVL C01334 V=800.0 PL=0
MOVL C01335 V=800.0 PL=0
MOVL C01336 V=800.0 PL=0
MOVL C01337 V=800.0 PL=0
MOVL C01338 V=800.0 PL=0
MOVL C01339 V=800.0 PL=0
MOVL C01340 V=800.0 PL=0
MOVL C01341 V=800.0 PL=0
MOVL C01342 V=800.0 PL=0
MOVL C01343 V=800.0 PL=0
MOVL C01344 V=800.0 PL=0
MOVL C01345 V=800.0 PL=0
MOVL C01346 V=800.0 PL=0
MOVL C01347 V=800.0 PL=0
MOVL C01348 V=800.0 PL=0
MOVL C01349 V=800.0 PL=0
MOVL C01350 V=800.0 PL=0
MOVL C01351 V=800.0 PL=0
MOVL C01352 V=800.0 PL=0
MOVL C01353 V=800.0 PL=0
MOVL C01354 V=800.0 PL=0
MOVL C01355 V=800.0 PL=0
MOVL C01356 V=800.0 PL=0
MOVL C01357 V=800.0 PL=0
MOVL C01358 V=800.0 PL=0
MOVL C01359 V=800.0 PL=0
MOVL C01360 V=800.0 PL=0
MOVL C01361 V=800.0 PL=0
MOVL C01362 V=800.0 PL=0
MOVL C01363 V=800.0 PL=0
MOVL C01364 V=800.0 PL=0
MOVL C01365 V=800.0 PL=0
MOVL C01366 V=800.0 PL=0
MOVL C01367 V=800.0 PL=0
MOVL C01368 V=800.0 PL=0
MOVL C01369 V=800.0 PL=0
MOVL C01370 V=800.0 PL=0
MOVL C01371 V=800.0 PL=0
MOVL C01372 V=800.0 PL=0
MOVL C01373 V=800.0 PL=0
MOVL C01374 V=800.0 PL=0
MOVL C01375 V=800.0 PL=0
MOVL C01376 V=800.0 PL=0
MOVL C01377 V=800.0 PL=0
MOVL C01378 V=800.0 PL=0
MOVL C01379 V=800.0 PL=0
MOVL C01380 V=800.0 PL=0
MOVL C01381 V=800.0 PL=0
MOVL C01382 V=800.0 PL=0
MOVL C01383 V=800.0 PL=0
MOVL C01384 V=800.0 PL=0
MOVL C01385 V=800.0 PL=0
MOVL C01386 V=800.0 PL=0
MOVL C01387 V=800.0 PL=0
MOVL C01388 V=800.0 PL=0
MOVL C01389 V=800.0 PL=0
MOVL C01390 V=800.0 PL=0
MOVL C01391 V=800.0 PL=0
MOVL C01392 V=800.0 PL=0
MOVL C01393 V=800.0 PL=0
MOVL C01394 V=800.0 PL=0
MOVL C01395 V=800.0 PL=0
MOVL C01396 V=800.0 PL=0
MOVL C01397 V=800.0 PL=0
MOVL C01398 V=800.0 PL=0
MOVL C01399 V=800.0 PL=0
MOVL C01400 V=800.0 PL=0
MOVL C01401 V=800.0 PL=0
MOVL C01402 V=800.0 PL=0
MOVL C01403 V=800.0 PL=0
MOVL C01404 V=800.0 PL=0
MOVL C01405 V=800.0 PL=0
MOVL C01406 V=800.0 PL=0
MOVL C01407 V=800.0 PL=0
MOVL C01408 V=800.0 PL=0
MOVL C01409 V=800.0 PL=0
MOVL C01410 V=800.0 PL=0
MOVL C01411 V=800.0 PL=0
MOVL C01412 V=800.0 PL=0
MOVL C01413 V=800.0 PL=0
MOVL C01414 V=800.0 PL=0
MOVL C01415 V=800.0 PL=0
MOVL C01416 V=800.0 PL=0
MOVL C01417 V=800.0 PL=0
MOVL C01418 V=800.0 PL=0
MOVL C01419 V=800.0 PL=0
MOVL C01420 V=800.0 PL=0
MOVL C01421 V=800.0 PL=0
MOVL C01422 V=800.0 PL=0
MOVL C01423 V=800.0 PL=0
MOVL C01424 V=800.0 PL=0
MOVL C01425 V=800.0 PL=0
MOVL C01426 V=800.0 PL=0
MOVL C01427 V=800.0 PL=0
MOVL C01428 V=800.0 PL=0
MOVL C01429 V=800.0 PL=0
MOVL C01430 V=800.0 PL=0
MOVL C01431 V=800.0 PL=0
MOVL C01432 V=800.0 PL=0
MOVL C01433 V=800.0 PL=0
MOVL C01434 V=800.0 PL=0
MOVL C01435 V=800.0 PL=0
MOVL C01436 V=800.0 PL=0
MOVL C01437 V=800.0 PL=0
MOVL C01438 V=800.0 PL=0
MOVL C01439 V=800.0 PL=0
MOVL C01440 V=800.0 PL=0
MOVL C01441 V=800.0 PL=0
MOVL C01442 V=800.0 PL=0
MOVL C01443 V=800.0 PL=0
MOVL C01444 V=800.0 PL=0
MOVL C01445 V=800.0 PL=0
MOVL C01446 V=800.0 PL=0
MOVL C01447 V=800.0 PL=0
MOVL C01448 V=800.0 PL=0
MOVL C01449 V=800.0 PL=0
MOVL C01450 V=800.0 PL=0
MOVL C01451 V=800.0 PL=0
MOVL C01452 V=800.0 PL=0
MOVL C01453 V=800.0 PL=0
MOVL C01454 V=800.0 PL=0
MOVL C01455 V=800.0 PL=0
MOVL C01456 V=800.0 PL=0
MOVL C01457 V=800.0 PL=0
MOVL C01458 V=800.0 PL=0
MOVL C01459 V=800.0 PL=0
MOVL C01460 V=800.0 PL=0
MOVL C01461 V=800.0 PL=0
MOVL C01462 V=800.0 PL=0
MOVL C01463 V=800.0 PL=0
MOVL C01464 V=800.0 PL=0
MOVL C01465 V=800.0 PL=0
MOVL C01466 V=800.0 PL=0
MOVL C01467 V=800.0 PL=0
MOVL C01468 V=800.0 PL=0
MOVL C01469 V=800.0 PL=0
MOVL C01470 V=800.0 PL=0
MOVL C01471 V=800.0 PL=0
MOVL C01472 V=800.0 PL=0
MOVL C01473 V=800.0 PL=0
MOVL C01474 V=800.0 PL=0
MOVL C01475 V=800.0 PL=0
MOVL C01476 V=800.0 PL=0
MOVL C01477 V=800.0 PL=0
MOVL C01478 V=800.0 PL=0
MOVL C01479 V=800.0 PL=0
MOVL C01480 V=800.0 PL=0
MOVL C01481 V=800.0 PL=0
MOVL C01482 V=800.0 PL=0
MOVL C01483 V=800.0 PL=0
MOVL C01484 V=800.0 PL=0
MOVL C01485 V=800.0 PL=0
MOVL C01486 V=800.0 PL=0
MOVL C01487 V=800.0 PL=0
MOVL C01488 V=800.0 PL=0
MOVL C01489 V=800.0 PL=0
MOVL C01490 V=800.0 PL=0
MOVL C01491 V=800.0 PL=0
MOVL C01492 V=800.0 PL=0
MOVL C01493 V=800.0 PL=0
MOVL C01494 V=800.0 PL=0
MOVL C01495 V=800.0 PL=0
MOVL C01496 V=800.0 PL=0
MOVL C01497 V=800.0 PL=0
MOVL C01498 V=800.0 PL=0
MOVL C01499 V=800.0 PL=0
MOVL C01500 V=800.0 PL=0
MOVL C01501 V=800.0 PL=0
MOVL C01502 V=800.0 PL=0
MOVL C01503 V=800.0 PL=0
MOVL C01504 V=800.0 PL=0
MOVL C01505 V=800.0 PL=0
MOVL C01506 V=800.0 PL=0
MOVL C01507 V=800.0 PL=0
MOVL C01508 V=800.0 PL=0
MOVL C01509 V=800.0 PL=0
MOVL C01510 V=800.0 PL=0
MOVL C01511 V=800.0 PL=0
MOVL C01512 V=800.0 PL=0
MOVL C01513 V=800.0 PL=0
MOVL C01514 V=800.0 PL=0
MOVL C01515 V=800.0 PL=0
MOVL C01516 V=800.0 PL=0
MOVL C01517 V=800.0 PL=0
MOVL C01518 V=800.0 PL=0
MOVL C01519 V=800.0 PL=0
MOVL C01520 V=800.0 PL=0
MOVL C01521 V=800.0 PL=0
MOVL C01522 V=800.0 PL=0
MOVL C01523 V=800.0 PL=0
MOVL C01524 V=800.0 PL=0
MOVL C01525 V=800.0 PL=0
MOVL C01526 V=800.0 PL=0
MOVL C01527 V=800.0 PL=0
MOVL C01528 V=800.0 PL=0
MOVL C01529 V=800.0 PL=0
MOVL C01530 V=800.0 PL=0
MOVL C01531 V=800.0 PL=0
MOVL C01532 V=800.0 PL=0
MOVL C01533 V=800.0 PL=0
MOVL C01534 V=800.0 PL=0
MOVL C01535 V=800.0 PL=0
MOVL C01536 V=800.0 PL=0
MOVL C01537 V=800.0 PL=0
MOVL C01538 V=800.0 PL=0
MOVL C01539 V=800.0 PL=0
MOVL C01540 V=800.0 PL=0
MOVL C01541 V=800.0 PL=0
MOVL C01542 V=800.0 PL=0
MOVL C01543 V=800.0 PL=0
MOVL C01544 V=800.0 PL=0
MOVL C01545 V=800.0 PL=0
MOVL C01546 V=800.0 PL=0
MOVL C01547 V=800.0 PL=0
MOVL C01548 V=800.0 PL=0
MOVL C01549 V=800.0 PL=0
MOVL C01550 V=800.0 PL=0
MOVL C01551 V=800.0 PL=0
MOVL C01552 V=800.0 PL=0
MOVL C01553 V=800.0 PL=0
MOVL C01554 V=800.0 PL=0
MOVL C01555 V=800.0 PL=0
MOVL C01556 V=800.0 PL=0
MOVL C01557 V=800.0 PL=0
MOVL C01558 V=800.0 PL=0
MOVL C01559 V=800.0 PL=0
MOVL C01560 V=800.0 PL=0
MOVL C01561 V=800.0 PL=0
MOVL C01562 V=800.0 PL=0
MOVL C01563 V=800.0 PL=0
MOVL C01564 V=800.0 PL=0
MOVL C01565 V=800.0 PL=0
MOVL C01566 V=800.0 PL=0
MOVL C01567 V=800.0 PL=0
MOVL C01568 V=800.0 PL=0
MOVL C01569 V=800.0 PL=0
MOVL C01570 V=800.0 PL=0
MOVL C01571 V=800.0 PL=0
MOVL C01572 V=800.0 PL=0
MOVL C01573 V=800.0 PL=0
MOVL C01574 V=800.0 PL=0
MOVL C01575 V=800.0 PL=0
MOVL C01576 V=800.0 PL=0
MOVL C01577 V=800.0 PL=0
MOVL C01578 V=800.0 PL=0
MOVL C01579 V=800.0 PL=0
MOVL C01580 V=800.0 PL=0
MOVL C01581 V=800.0 PL=0
MOVL C01582 V=800.0 PL=0
MOVL C01583 V=800.0 PL=0
MOVL C01584 V=800.0 PL=0
MOVL C01585 V=800.0 PL=0
MOVL C01586 V=800.0 PL=0
MOVL C01587 V=800.0 PL=0
MOVL C01588 V=800.0 PL=0
MOVL C01589 V=800.0 PL=0
MOVL C01590 V=800.0 PL=0
MOVL C01591 V=800.0 PL=0
MOVL C01592 V=800.0 PL=0
MOVL C01593 V=800.0 PL=0
MOVL C01594 V=800.0 PL=0
MOVL C01595 V=800.0 PL=0
MOVL C01596 V=800.0 PL=0
MOVL C01597 V=800.0 PL=0
MOVL C01598 V=800.0 PL=0
MOVL C01599 V=800.0 PL=0
MOVL C01600 V=800.0 PL=0
MOVL C01601 V=800.0 PL=0
MOVL C01602 V=800.0 PL=0
MOVL C01603 V=800.0 PL=0
MOVL C01604 V=800.0 PL=0
MOVL C01605 V=800.0 PL=0
MOVL C01606 V=800.0 PL=0
MOVL C01607 V=800.0 PL=0
MOVL C01608 V=800.0 PL=0
MOVL C01609 V=800.0 PL=0
MOVL C01610 V=800.0 PL=0
MOVL C01611 V=800.0 PL=0
MOVL C01612 V=800.0 PL=0
MOVL C01613 V=800.0 PL=0
MOVL C01614 V=800.0 PL=0
MOVL C01615 V=800.0 PL=0
MOVL C01616 V=800.0 PL=0
MOVL C01617 V=800.0 PL=0
MOVL C01618 V=800.0 PL=0
MOVL C01619 V=800.0 PL=0
MOVL C01620 V=800.0 PL=0
MOVL C01621 V=800.0 PL=0
MOVL C01622 V=800.0 PL=0
MOVL C01623 V=800.0 PL=0
MOVL C01624 V=800.0 PL=0
MOVL C01625 V=800.0 PL=0
MOVL C01626 V=800.0 PL=0
MOVL C01627 V=800.0 PL=0
MOVL C01628 V=800.0 PL=0
MOVL C01629 V=800.0 PL=0
MOVL C01630 V=800.0 PL=0
MOVL C01631 V=800.0 PL=0
MOVL C01632 V=800.0 PL=0
MOVL C01633 V=800.0 PL=0
MOVL C01634 V=800.0 PL=0
MOVL C01635 V=800.0 PL=0
MOVL C01636 V=800.0 PL=0
MOVL C01637 V=800.0 PL=0
MOVL C01638 V=800.0 PL=0
MOVL C01639 V=800.0 PL=0
MOVL C01640 V=800.0 PL=0
MOVL C01641 V=800.0 PL=0
MOVL C01642 V=800.0 PL=0
MOVL C01643 V=800.0 PL=0
MOVL C01644 V=800.0 PL=0
MOVL C01645 V=800.0 PL=0
MOVL C01646 V=800.0 PL=0
MOVL C01647 V=800.0 PL=0
MOVL C01648 V=800.0 PL=0
MOVL C01649 V=800.0 PL=0
MOVL C01650 V=800.0 PL=0
MOVL C01651 V=800.0 PL=0
MOVL C01652 V=800.0 PL=0
MOVL C01653 V=800.0 PL=0
MOVL C01654 V=800.0 PL=0
MOVL C01655 V=800.0 PL=0
MOVL C01656 V=800.0 PL=0
MOVL C01657 V=800.0 PL=0
MOVL C01658 V=800.0 PL=0
MOVL C01659 V=800.0 PL=0
MOVL C01660 V=800.0 PL=0
MOVL C01661 V=800.0 PL=0
MOVL C01662 V=800.0 PL=0
MOVL C01663 V=800.0 PL=0
MOVL C01664 V=800.0 PL=0
MOVL C01665 V=800.0 PL=0
MOVL C01666 V=800.0 PL=0
MOVL C01667 V=800.0 PL=0
MOVL C01668 V=800.0 PL=0
MOVL C01669 V=800.0 PL=0
MOVL C01670 V=800.0 PL=0
MOVL C01671 V=800.0 PL=0
MOVL C01672 V=800.0 PL=0
MOVL C01673 V=800.0 PL=0
MOVL C01674 V=800.0 PL=0
MOVL C01675 V=800.0 PL=0
MOVL C01676 V=800.0 PL=0
MOVL C01677 V=800.0 PL=0
MOVL C01678 V=800.0 PL=0
MOVL C01679 V=800.0 PL=0
MOVL C01680 V=800.0 PL=0
MOVL C01681 V=800.0 PL=0
MOVL C01682 V=800.0 PL=0
MOVL C01683 V=800.0 PL=0
MOVL C01684 V=800.0 PL=0
MOVL C01685 V=800.0 PL=0
MOVL C01686 V=800.0 PL=0
MOVL C01687 V=800.0 PL=0
MOVL C01688 V=800.0 PL=0
MOVL C01689 V=800.0 PL=0
MOVL C01690 V=800.0 PL=0
MOVL C01691 V=800.0 PL=0
MOVL C01692 V=800.0 PL=0
MOVL C01693 V=800.0 PL=0
MOVL C01694 V=800.0 PL=0
MOVL C01695 V=800.0 PL=0
MOVL C01696 V=800.0 PL=0
MOVL C01697 V=800.0 PL=0
MOVL C01698 V=800.0 PL=0
MOVL C01699 V=800.0 PL=0
MOVL C01700 V=800.0 PL=0
MOVL C01701 V=800.0 PL=0
MOVL C01702 V=800.0 PL=0
MOVL C01703 V=800.0 PL=0
MOVL C01704 V=800.0 PL=0
MOVL C01705 V=800.0 PL=0
MOVL C01706 V=800.0 PL=0
MOVL C01707 V=800.0 PL=0
MOVL C01708 V=800.0 PL=0
MOVL C01709 V=800.0 PL=0
MOVL C01710 V=800.0 PL=0
MOVL C01711 V=800.0 PL=0
MOVL C01712 V=800.0 PL=0
MOVL C01713 V=800.0 PL=0
MOVL C01714 V=800.0 PL=0
MOVL C01715 V=800.0 PL=0
MOVL C01716 V=800.0 PL=0
MOVL C01717 V=800.0 PL=0
MOVL C01718 V=800.0 PL=0
MOVL C01719 V=800.0 PL=0
MOVL C01720 V=800.0 PL=0
MOVL C01721 V=800.0 PL=0
MOVL C01722 V=800.0 PL=0
MOVL C01723 V=800.0 PL=0
MOVL C01724 V=800.0 PL=0
MOVL C01725 V=800.0 PL=0
MOVL C01726 V=800.0 PL=0
MOVL C01727 V=800.0 PL=0
MOVL C01728 V=800.0 PL=0
MOVL C01729 V=800.0 PL=0
MOVL C01730 V=800.0 PL=0
MOVL C01731 V=800.0 PL=0
MOVL C01732 V=800.0 PL=0
MOVL C01733 V=800.0 PL=0
MOVL C01734 V=800.0 PL=0
MOVL C01735 V=800.0 PL=0
MOVL C01736 V=800.0 PL=0
MOVL C01737 V=800.0 PL=0
MOVL C01738 V=800.0 PL=0
MOVL C01739 V=800.0 PL=0
MOVL C01740 V=800.0 PL=0
MOVL C01741 V=800.0 PL=0
MOVL C01742 V=800.0 PL=0
MOVL C01743 V=800.0 PL=0
MOVL C01744 V=800.0 PL=0
MOVL C01745 V=800.0 PL=0
MOVL C01746 V=800.0 PL=0
MOVL C01747 V=800.0 PL=0
MOVL C01748 V=800.0 PL=0
MOVL C01749 V=800.0 PL=0
MOVL C01750 V=800.0 PL=0
MOVL C01751 V=800.0 PL=0
MOVL C01752 V=800.0 PL=0
MOVL C01753 V=800.0 PL=0
MOVL C01754 V=800.0 PL=0
MOVL C01755 V=800.0 PL=0
MOVL C01756 V=800.0 PL=0
MOVL C01757 V=800.0 PL=0
MOVL C01758 V=800.0 PL=0
MOVL C01759 V=800.0 PL=0
MOVL C01760 V=800.0 PL=0
MOVL C01761 V=800.0 PL=0
MOVL C01762 V=800.0 PL=0
MOVL C01763 V=800.0 PL=0
MOVL C01764 V=800.0 PL=0
MOVL C01765 V=800.0 PL=0
MOVL C01766 V=800.0 PL=0
MOVL C01767 V=800.0 PL=0
MOVL C01768 V=800.0 PL=0
MOVL C01769 V=800.0 PL=0
MOVL C01770 V=800.0 PL=0
MOVL C01771 V=800.0 PL=0
MOVL C01772 V=800.0 PL=0
MOVL C01773 V=800.0 PL=0
MOVL C01774 V=800.0 PL=0
MOVL C01775 V=800.0 PL=0
MOVL C01776 V=800.0 PL=0
MOVL C01777 V=800.0 PL=0
MOVL C01778 V=800.0 PL=0
MOVL C01779 V=800.0 PL=0
MOVL C01780 V=800.0 PL=0
MOVL C01781 V=800.0 PL=0
MOVL C01782 V=800.0 PL=0
MOVL C01783 V=800.0 PL=0
MOVL C01784 V=800.0 PL=0
MOVL C01785 V=800.0 PL=0
MOVL C01786 V=800.0 PL=0
MOVL C01787 V=800.0 PL=0
MOVL C01788 V=800.0 PL=0
MOVL C01789 V=800.0 PL=0
MOVL C01790 V=800.0 PL=0
MOVL C01791 V=800.0 PL=0
MOVL C01792 V=800.0 PL=0
MOVL C01793 V=800.0 PL=0
MOVL C01794 V=800.0 PL=0
MOVL C01795 V=800.0 PL=0
MOVL C01796 V=800.0 PL=0
MOVL C01797 V=800.0 PL=0
MOVL C01798 V=800.0 PL=0
MOVL C01799 V=800.0 PL=0
MOVL C01800 V=800.0 PL=0
MOVL C01801 V=800.0 PL=0
MOVL C01802 V=800.0 PL=0
MOVL C01803 V=800.0 PL=0
MOVL C01804 V=800.0 PL=0
MOVL C01805 V=800.0 PL=0
MOVL C01806 V=800.0 PL=0
MOVL C01807 V=800.0 PL=0
MOVL C01808 V=800.0 PL=0
MOVL C01809 V=800.0 PL=0
MOVL C01810 V=800.0 PL=0
MOVL C01811 V=800.0 PL=0
MOVL C01812 V=800.0 PL=0
MOVL C01813 V=800.0 PL=0
MOVL C01814 V=800.0 PL=0
MOVL C01815 V=800.0 PL=0
MOVL C01816 V=800.0 PL=0
MOVL C01817 V=800.0 PL=0
MOVL C01818 V=800.0 PL=0
MOVL C01819 V=800.0 PL=0
MOVL C01820 V=800.0 PL=0
MOVL C01821 V=800.0 PL=0
MOVL C01822 V=800.0 PL=0
MOVL C01823 V=800.0 PL=0
MOVL C01824 V=800.0 PL=0
MOVL C01825 V=800.0 PL=0
MOVL C01826 V=800.0 PL=0
MOVL C01827 V=800.0 PL=0
MOVL C01828 V=800.0 PL=0
MOVL C01829 V=800.0 PL=0
MOVL C01830 V=800.0 PL=0
MOVL C01831 V=800.0 PL=0
MOVL C01832 V=800.0 PL=0
MOVL C01833 V=800.0 PL=0
MOVL C01834 V=800.0 PL=0
MOVL C01835 V=800.0 PL=0
MOVL C01836 V=800.0 PL=0
MOVL C01837 V=800.0 PL=0
MOVL C01838 V=800.0 PL=0
MOVL C01839 V=800.0 PL=0
MOVL C01840 V=800.0 PL=0
MOVL C01841 V=800.0 PL=0
MOVL C01842 V=800.0 PL=0
MOVL C01843 V=800.0 PL=0
MOVL C01844 V=800.0 PL=0
MOVL C01845 V=800.0 PL=0
MOVL C01846 V=800.0 PL=0
MOVL C01847 V=800.0 PL=0
MOVL C01848 V=800.0 PL=0
MOVL C01849 V=800.0 PL=0
MOVL C01850 V=800.0 PL=0
MOVL C01851 V=800.0 PL=0
MOVL C01852 V=800.0 PL=0
MOVL C01853 V=800.0 PL=0
MOVL C01854 V=800.0 PL=0
MOVL C01855 V=800.0 PL=0
MOVL C01856 V=800.0 PL=0
MOVL C01857 V=800.0 PL=0
MOVL C01858 V=800.0 PL=0
MOVL C01859 V=800.0 PL=0
MOVL C01860 V=800.0 PL=0
MOVL C01861 V=800.0 PL=0
MOVL C01862 V=800.0 PL=0
MOVL C01863 V=800.0 PL=0
MOVL C01864 V=800.0 PL=0
MOVL C01865 V=800.0 PL=0
MOVL C01866 V=800.0 PL=0
MOVL C01867 V=800.0 PL=0
MOVL C01868 V=800.0 PL=0
MOVL C01869 V=800.0 PL=0
MOVL C01870 V=800.0 PL=0
MOVL C01871 V=800.0 PL=0
MOVL C01872 V=800.0 PL=0
MOVL C01873 V=800.0 PL=0
MOVL C01874 V=800.0 PL=0
MOVL C01875 V=800.0 PL=0
MOVL C01876 V=800.0 PL=0
MOVL C01877 V=800.0 PL=0
MOVL C01878 V=800.0 PL=0
MOVL C01879 V=800.0 PL=0
MOVL C01880 V=800.0 PL=0
MOVL C01881 V=800.0 PL=0
MOVL C01882 V=800.0 PL=0
MOVL C01883 V=800.0 PL=0
MOVL C01884 V=800.0 PL=0
MOVL C01885 V=800.0 PL=0
MOVL C01886 V=800.0 PL=0
MOVL C01887 V=800.0 PL=0
MOVL C01888 V=800.0 PL=0
MOVL C01889 V=800.0 PL=0
MOVL C01890 V=800.0 PL=0
MOVL C01891 V=800.0 PL=0
MOVL C01892 V=800.0 PL=0
MOVL C01893 V=800.0 PL=0
MOVL C01894 V=800.0 PL=0
MOVL C01895 V=800.0 PL=0
MOVL C01896 V=800.0 PL=0
MOVL C01897 V=800.0 PL=0
MOVL C01898 V=800.0 PL=0
MOVL C01899 V=800.0 PL=0
MOVL C01900 V=800.0 PL=0
MOVL C01901 V=800.0 PL=0
MOVL C01902 V=800.0 PL=0
MOVL C01903 V=800.0 PL=0
MOVL C01904 V=800.0 PL=0
MOVL C01905 V=800.0 PL=0
MOVL C01906 V=800.0 PL=0
MOVL C01907 V=800.0 PL=0
MOVL C01908 V=800.0 PL=0
MOVL C01909 V=800.0 PL=0
MOVL C01910 V=800.0 PL=0
MOVL C01911 V=800.0 PL=0
MOVL C01912 V=800.0 PL=0
MOVL C01913 V=800.0 PL=0
MOVL C01914 V=800.0 PL=0
MOVL C01915 V=800.0 PL=0
MOVL C01916 V=800.0 PL=0
MOVL C01917 V=800.0 PL=0
MOVL C01918 V=800.0 PL=0
MOVL C01919 V=800.0 PL=0
MOVL C01920 V=800.0 PL=0
MOVL C01921 V=800.0 PL=0
MOVL C01922 V=800.0 PL=0
MOVL C01923 V=800.0 PL=0
MOVL C01924 V=800.0 PL=0
MOVL C01925 V=800.0 PL=0
MOVL C01926 V=800.0 PL=0
MOVL C01927 V=800.0 PL=0
MOVL C01928 V=800.0 PL=0
MOVL C01929 V=800.0 PL=0
MOVL C01930 V=800.0 PL=0
MOVL C01931 V=800.0 PL=0
MOVL C01932 V=800.0 PL=0
MOVL C01933 V=800.0 PL=0
MOVL C01934 V=800.0 PL=0
MOVL C01935 V=800.0 PL=0
MOVL C01936 V=800.0 PL=0
MOVL C01937 V=800.0 PL=0
MOVL C01938 V=800.0 PL=0
MOVL C01939 V=800.0 PL=0
MOVL C01940 V=800.0 PL=0
MOVL C01941 V=800.0 PL=0
MOVL C01942 V=800.0 PL=0
MOVL C01943 V=800.0 PL=0
MOVL C01944 V=800.0 PL=0
MOVL C01945 V=800.0 PL=0
MOVL C01946 V=800.0 PL=0
MOVL C01947 V=800.0 PL=0
MOVL C01948 V=800.0 PL=0
MOVL C01949 V=800.0 PL=0
MOVL C01950 V=800.0 PL=0
MOVL C01951 V=800.0 PL=0
MOVL C01952 V=800.0 PL=0
MOVL C01953 V=800.0 PL=0
MOVL C01954 V=800.0 PL=0
MOVL C01955 V=800.0 PL=0
MOVL C01956 V=800.0 PL=0
MOVL C01957 V=800.0 PL=0
MOVL C01958 V=800.0 PL=0
MOVL C01959 V=800.0 PL=0
MOVL C01960 V=800.0 PL=0
MOVL C01961 V=800.0 PL=0
MOVL C01962 V=800.0 PL=0
MOVL C01963 V=800.0 PL=0
MOVL C01964 V=800.0 PL=0
MOVL C01965 V=800.0 PL=0
MOVL C01966 V=800.0 PL=0
MOVL C01967 V=800.0 PL=0
MOVL C01968 V=800.0 PL=0
MOVL C01969 V=800.0 PL=0
MOVL C01970 V=800.0 PL=0
MOVL C01971 V=800.0 PL=0
MOVL C01972 V=800.0 PL=0
MOVL C01973 V=800.0 PL=0
MOVL C01974 V=800.0 PL=0
MOVL C01975 V=800.0 PL=0
MOVL C01976 V=800.0 PL=0
MOVL C01977 V=800.0 PL=0
MOVL C01978 V=800.0 PL=0
MOVL C01979 V=800.0 PL=0
MOVL C01980 V=800.0 PL=0
MOVL C01981 V=800.0 PL=0
MOVL C01982 V=800.0 PL=0
MOVL C01983 V=800.0 PL=0
MOVL C01984 V=800.0 PL=0
MOVL C01985 V=800.0 PL=0
MOVL C01986 V=800.0 PL=0
MOVL C01987 V=800.0 PL=0
MOVL C01988 V=800.0 PL=0
MOVL C01989 V=800.0 PL=0
MOVL C01990 V=800.0 PL=0
MOVL C01991 V=800.0 PL=0
MOVL C01992 V=800.0 PL=0
MOVL C01993 V=800.0 PL=0
MOVL C01994 V=800.0 PL=0
MOVL C01995 V=800.0 PL=0
MOVL C01996 V=800.0 PL=0
MOVL C01997 V=800.0 PL=0
MOVL C01998 V=800.0 PL=0
MOVL C01999 V=800.0 PL=0
MOVL C02000 V=800.0 PL=0
MOVL C02001 V=800.0 PL=0
MOVL C02002 V=800.0 PL=0
MOVL C02003 V=800.0 PL=0
MOVL C02004 V=800.0 PL=0
MOVL C02005 V=800.0 PL=0
MOVL C02006 V=800.0 PL=0
MOVL C02007 V=800.0 PL=0
MOVL C02008 V=800.0 PL=0
MOVL C02009 V=800.0 PL=0
MOVL C02010 V=800.0 PL=0
MOVL C02011 V=800.0 PL=0
MOVL C02012 V=800.0 PL=0
MOVL C02013 V=800.0 PL=0
MOVL C02014 V=800.0 PL=0
MOVL C02015 V=800.0 PL=0
MOVL C02016 V=800.0 PL=0
MOVL C02017 V=800.0 PL=0
MOVL C02018 V=800.0 PL=0
MOVL C02019 V=800.0 PL=0
MOVL C02020 V=800.0 PL=0
MOVL C02021 V=800.0 PL=0
MOVL C02022 V=800.0 PL=0
MOVL C02023 V=800.0 PL=0
MOVL C02024 V=800.0 PL=0
MOVL C02025 V=800.0 PL=0
MOVL C02026 V=800.0 PL=0
MOVL C02027 V=800.0 PL=0
MOVL C02028 V=800.0 PL=0
MOVL C02029 V=800.0 PL=0
MOVL C02030 V=800.0 PL=0
MOVL C02031 V=800.0 PL=0
MOVL C02032 V=800.0 PL=0
MOVL C02033 V=800.0 PL=0
MOVL C02034 V=800.0 PL=0
MOVL C02035 V=800.0 PL=0
MOVL C02036 V=800.0 PL=0
MOVL C02037 V=800.0 PL=0
MOVL C02038 V=800.0 PL=0
MOVL C02039 V=800.0 PL=0
MOVL C02040 V=800.0 PL=0
MOVL C02041 V=800.0 PL=0
MOVL C02042 V=800.0 PL=0
MOVL C02043 V=800.0 PL=0
MOVL C02044 V=800.0 PL=0
MOVL C02045 V=800.0 PL=0
MOVL C02046 V=800.0 PL=0
MOVL C02047 V=800.0 PL=0
MOVL C02048 V=800.0 PL=0
MOVL C02049 V=800.0 PL=0
MOVL C02050 V=800.0 PL=0
MOVL C02051 V=800.0 PL=0
MOVL C02052 V=800.0 PL=0
MOVL C02053 V=800.0 PL=0
MOVL C02054 V=800.0 PL=0
MOVL C02055 V=800.0 PL=0
MOVL C02056 V=800.0 PL=0
MOVL C02057 V=800.0 PL=0
MOVL C02058 V=800.0 PL=0
MOVL C02059 V=800.0 PL=0
MOVL C02060 V=800.0 PL=0
MOVL C02061 V=800.0 PL=0
MOVL C02062 V=800.0 PL=0
MOVL C02063 V=800.0 PL=0
MOVL C02064 V=800.0 PL=0
MOVL C02065 V=800.0 PL=0
MOVL C02066 V=800.0 PL=0
MOVL C02067 V=800.0 PL=0
MOVL C02068 V=800.0 PL=0
MOVL C02069 V=800.0 PL=0
MOVL C02070 V=800.0 PL=0
MOVL C02071 V=800.0 PL=0
MOVL C02072 V=800.0 PL=0
MOVL C02073 V=800.0 PL=0
MOVL C02074 V=800.0 PL=0
MOVL C02075 V=800.0 PL=0
MOVL C02076 V=800.0 PL=0
MOVL C02077 V=800.0 PL=0
MOVL C02078 V=800.0 PL=0
MOVL C02079 V=800.0 PL=0
MOVL C02080 V=800.0 PL=0
MOVL C02081 V=800.0 PL=0
MOVL C02082 V=800.0 PL=0
MOVL C02083 V=800.0 PL=0
MOVL C02084 V=800.0 PL=0
MOVL C02085 V=800.0 PL=0
MOVL C02086 V=800.0 PL=0
MOVL C02087 V=800.0 PL=0
MOVL C02088 V=800.0 PL=0
MOVL C02089 V=800.0 PL=0
MOVL C02090 V=800.0 PL=0
MOVL C02091 V=800.0 PL=0
MOVL C02092 V=800.0 PL=0
MOVL C02093 V=800.0 PL=0
MOVL C02094 V=800.0 PL=0
MOVL C02095 V=800.0 PL=0
MOVL C02096 V=800.0 PL=0
MOVL C02097 V=800.0 PL=0
MOVL C02098 V=800.0 PL=0
MOVL C02099 V=800.0 PL=0
MOVL C02100 V=800.0 PL=0
MOVL C02101 V=800.0 PL=0
MOVL C02102 V=800.0 PL=0
MOVL C02103 V=800.0 PL=0
MOVL C02104 V=800.0 PL=0
MOVL C02105 V=800.0 PL=0
MOVL C02106 V=800.0 PL=0
MOVL C02107 V=800.0 PL=0
MOVL C02108 V=800.0 PL=0
MOVL C02109 V=800.0 PL=0
MOVL C02110 V=800.0 PL=0
MOVL C02111 V=800.0 PL=0
MOVL C02112 V=800.0 PL=0
MOVL C02113 V=800.0 PL=0
MOVL C02114 V=800.0 PL=0
MOVL C02115 V=800.0 PL=0
MOVL C02116 V=800.0 PL=0
MOVL C02117 V=800.0 PL=0
MOVL C02118 V=800.0 PL=0
MOVL C02119 V=800.0 PL=0
MOVL C02120 V=800.0 PL=0
MOVL C02121 V=800.0 PL=0
MOVL C02122 V=800.0 PL=0
MOVL C02123 V=800.0 PL=0
MOVL C02124 V=800.0 PL=0
MOVL C02125 V=800.0 PL=0
MOVL C02126 V=800.0 PL=0
MOVL C02127 V=800.0 PL=0
MOVL C02128 V=800.0 PL=0
MOVL C02129 V=800.0 PL=0
MOVL C02130 V=800.0 PL=0
MOVL C02131 V=800.0 PL=0
MOVL C02132 V=800.0 PL=0
MOVL C02133 V=800.0 PL=0
MOVL C02134 V=800.0 PL=0
MOVL C02135 V=800.0 PL=0
MOVL C02136 V=800.0 PL=0
MOVL C02137 V=800.0 PL=0
MOVL C02138 V=800.0 PL=0
MOVL C02139 V=800.0 PL=0
MOVL C02140 V=800.0 PL=0
MOVL C02141 V=800.0 PL=0
